               IF NOT "IX_HBW_SwitchCantileverFront_I5" AND "IX_HBW_SwitchCantileverBack_I6" THEN
                   IF "gtyp_VGR".x_HBW_Storage THEN
                       "gtyp_HBW".Rack_Workpiece[#li_Counter_Act_Ver, #li_Counter_Act_Hor].s_id := '';
                   ELSIF "gtyp_VGR".x_HBW_Outsource THEN
                       "gtyp_Interface_Dashboard".Subscribe.State_HBW.x_active := TRUE;
                       "gtyp_HBW".History := "gtyp_HBW".Rack_History[#li_Counter_Act_Ver, #li_Counter_Act_Hor].History;
                       "gtyp_HBW".Workpiece := "gtyp_HBW".Rack_Workpiece[#li_Counter_Act_Ver, #li_Counter_Act_Hor];
                       #li_Return_LDT := RD_SYS_T(#ldt_MQTT);
                       "gtyp_HBW".History[4].i_code := 400;
                       "gtyp_HBW".History[4].ldt_ts := DT_TO_LDT(#ldt_MQTT);

                       "gtyp_HBW".Rack_Workpiece[#li_Counter_Act_Ver, #li_Counter_Act_Hor].s_id := '';
                       "gtyp_HBW".Rack_Workpiece[#li_Counter_Act_Ver, #li_Counter_Act_Hor].s_state := '';
                       "gtyp_HBW".Rack_Workpiece[#li_Counter_Act_Ver, #li_Counter_Act_Hor].s_type := '';
                       FOR #li_Counter := 1 TO 8 DO
                           "gtyp_HBW".Rack_History[#li_Counter_Act_Ver, #li_Counter_Act_Hor].History[#li_Counter].i_code := 0;
                           "gtyp_HBW".Rack_History[#li_Counter_Act_Ver, #li_Counter_Act_Hor].History[#li_Counter].ldt_ts := DT#1990-01-01-00:00:00;
                       END_FOR;
                   END_IF;
                   "QX_HBW_M4_CantileverBackward_Q8" := FALSE;
                   "QX_HBW_M4_CantileverForward_Q7" := FALSE;
                   #li_StepCase := 110;
               END_IF;

           110: // homing vertical/horizontal axis

               "gtyp_HBW".Horizontal_Axis.x_Reference := TRUE;

               "gtyp_HBW".Vertical_Axis.di_Target_Position := "gtyp_HBW".di_PosBelt_Vertical - "gtyp_HBW".di_Offset_Pos_Belt_Vertical;
               "gtyp_HBW".Vertical_Axis.x_Start_Positioning := TRUE;

               IF ("gtyp_HBW".Vertical_Axis.di_Actual_Position <= ("gtyp_HBW".di_PosBelt_Vertical - "gtyp_HBW".di_Offset_Pos_Belt_Vertical + "gtyp_HBW".Vertical_Axis.Config.di_Pos_Window))
                   AND ("gtyp_HBW".Vertical_Axis.di_Actual_Position >= ("gtyp_HBW".di_PosBelt_Vertical - "gtyp_HBW".di_Offset_Pos_Belt_Vertical - "gtyp_HBW".Vertical_Axis.Config.di_Pos_Window))
                   AND "gtyp_HBW".Vertical_Axis.x_Position_Reached THEN
                   "gtyp_HBW".Vertical_Axis.x_Start_Positioning := FALSE;
               END_IF;

               IF NOT "gtyp_HBW".Horizontal_Axis.x_Referenced THEN
                   #li_StepCase := 120;
               END_IF;

           120: //homed vertical/horizontal axis

               IF "gtyp_HBW".Horizontal_Axis.x_Referenced THEN
                   "gtyp_HBW".Horizontal_Axis.x_Reference := FALSE;
               END_IF;

               IF ("gtyp_HBW".Vertical_Axis.di_Actual_Position <= ("gtyp_HBW".di_PosBelt_Vertical - "gtyp_HBW".di_Offset_Pos_Belt_Vertical + "gtyp_HBW".Vertical_Axis.Config.di_Pos_Window))
                   AND ("gtyp_HBW".Vertical_Axis.di_Actual_Position >= ("gtyp_HBW".di_PosBelt_Vertical - "gtyp_HBW".di_Offset_Pos_Belt_Vertical - "gtyp_HBW".Vertical_Axis.Config.di_Pos_Window))
                   AND "gtyp_HBW".Vertical_Axis.x_Position_Reached THEN
                   "gtyp_HBW".Vertical_Axis.x_Start_Positioning := FALSE;
               END_IF;

               IF "gtyp_HBW".Horizontal_Axis.x_Referenced
                   AND ("gtyp_HBW".Vertical_Axis.di_Actual_Position <= ("gtyp_HBW".di_PosBelt_Vertical - "gtyp_HBW".di_Offset_Pos_Belt_Vertical + "gtyp_HBW".Vertical_Axis.Config.di_Pos_Window))
                   AND ("gtyp_HBW".Vertical_Axis.di_Actual_Position >= ("gtyp_HBW".di_PosBelt_Vertical - "gtyp_HBW".di_Offset_Pos_Belt_Vertical - "gtyp_HBW".Vertical_Axis.Config.di_Pos_Window))
                   AND "gtyp_HBW".Vertical_Axis.x_Position_Reached THEN
                   "gtyp_HBW".Horizontal_Axis.x_Reference := FALSE;
                   "gtyp_HBW".Vertical_Axis.x_Start_Positioning := FALSE;
                   #li_StepCase := 130;
               END_IF;

           130: // Position vertical+offset/horizontal Belt
               "gtyp_HBW".Horizontal_Axis.di_Target_Position := "gtyp_HBW".di_PosBelt_Horizontal;
               "gtyp_HBW".Horizontal_Axis.x_Start_Positioning := TRUE;

               IF ("gtyp_HBW".Horizontal_Axis.di_Actual_Position <= ("gtyp_HBW".di_PosBelt_Horizontal + "gtyp_HBW".Horizontal_Axis.Config.di_Pos_Window))
                   AND ("gtyp_HBW".Horizontal_Axis.di_Actual_Position >= ("gtyp_HBW".di_PosBelt_Horizontal - "gtyp_HBW".Horizontal_Axis.Config.di_Pos_Window))
                   AND "gtyp_HBW".Horizontal_Axis.x_Position_Reached THEN
                   "gtyp_HBW".Horizontal_Axis.x_Start_Positioning := FALSE;
               END_IF;

               IF ("gtyp_HBW".Horizontal_Axis.di_Actual_Position <= ("gtyp_HBW".di_PosBelt_Horizontal + "gtyp_HBW".Horizontal_Axis.Config.di_Pos_Window))
                   AND ("gtyp_HBW".Horizontal_Axis.di_Actual_Position >= ("gtyp_HBW".di_PosBelt_Horizontal - "gtyp_HBW".Horizontal_Axis.Config.di_Pos_Window))
                   AND "gtyp_HBW".Horizontal_Axis.x_Position_Reached THEN
                   "gtyp_HBW".Horizontal_Axis.x_Start_Positioning := FALSE;
                   #li_StepCase := 140;
               END_IF;

           140: // Position cantilever Forward Belt

               "QX_HBW_M4_CantileverBackward_Q8" := FALSE;
               "QX_HBW_M4_CantileverForward_Q7" := TRUE;

               #lx_Time_Error := TRUE;

               IF "IX_HBW_SwitchCantileverFront_I5" AND NOT "IX_HBW_SwitchCantileverBack_I6" THEN
                   "QX_HBW_M4_CantileverBackward_Q8" := FALSE;
                   "QX_HBW_M4_CantileverForward_Q7" := FALSE;
                   #lx_Time_Error := FALSE;
                   #li_StepCase := 150;
               END_IF;

               // runtime error
               IF #lfb_TON_Error.Q THEN
                   #li_Lights := 4;
                   #lx_Time_Error := FALSE;
                   "QX_HBW_M1_ConveyorBeltBackward_Q2" := FALSE;
                   "QX_HBW_M1_ConveyorBeltForward_Q1" := FALSE;
                   "gtyp_Interface_Dashboard".Subscribe.State_HBW.x_active := FALSE;
                   "gtyp_HBW".x_Error := TRUE;
                   #li_StepCase := 0;
               END_IF;

           150: // Position vertical Belt
               "gtyp_HBW".Vertical_Axis.di_Target_Position := "gtyp_HBW".di_PosBelt_Vertical;
               "gtyp_HBW".Vertical_Axis.x_Start_Positioning := TRUE;

               IF ("gtyp_HBW".Vertical_Axis.di_Actual_Position <= ("gtyp_HBW".di_PosBelt_Vertical + "gtyp_HBW".Vertical_Axis.Config.di_Pos_Window))
                   AND ("gtyp_HBW".Vertical_Axis.di_Actual_Position >= ("gtyp_HBW".di_PosBelt_Vertical - "gtyp_HBW".Vertical_Axis.Config.di_Pos_Window))
                   AND "gtyp_HBW".Vertical_Axis.x_Position_Reached THEN
                   "gtyp_HBW".Vertical_Axis.x_Start_Positioning := FALSE;
                   #li_StepCase := 160;
               END_IF;

           160: // Start Conveyor Belt Forward

               #lx_Time_Error := TRUE;

               IF NOT "IX_HBW_LightBarrierInside_I2" THEN
                   "QX_HBW_M1_ConveyorBeltBackward_Q2" := FALSE;
                   "QX_HBW_M1_ConveyorBeltForward_Q1" := TRUE;
                   #lx_Time_Error := FALSE;
                   #li_StepCase := 170;
               END_IF;

               // runtime error
               IF #lfb_TON_Error.Q THEN
                   #li_Lights := 4;
                   #lx_Time_Error := FALSE;
                   "QX_HBW_M1_ConveyorBeltBackward_Q2" := FALSE;
                   "QX_HBW_M1_ConveyorBeltForward_Q1" := FALSE;
                   "gtyp_Interface_Dashboard".Subscribe.State_HBW.x_active := FALSE;
                   "gtyp_HBW".x_Error := TRUE;
                   #li_StepCase := 0;
               END_IF;

           170: //Run-on time reached Conveyor Belt Outside

               #lx_Time_Error := TRUE;

               IF #lfb_TON_ConveyerBelt_Out.Q THEN
                   "QX_HBW_M1_ConveyorBeltBackward_Q2" := FALSE;
                   "QX_HBW_M1_ConveyorBeltForward_Q1" := FALSE;
                   "gtyp_HBW".x_HBW_Container_Available := TRUE;
                   #lx_Time_Error := FALSE;
                   #li_StepCase := 180;
               END_IF;

               // runtime error
               IF #lfb_TON_Error.Q THEN
                   #li_Lights := 4;
                   #lx_Time_Error := FALSE;
                   "QX_HBW_M1_ConveyorBeltBackward_Q2" := FALSE;
                   "QX_HBW_M1_ConveyorBeltForward_Q1" := FALSE;
                   "gtyp_Interface_Dashboard".Subscribe.State_HBW.x_active := FALSE;
                   "gtyp_HBW".x_Error := TRUE;
                   #li_StepCase := 0;
               END_IF;

           180: // VGR picked up - outsource

               #li_Lights := 1;

               IF "gtyp_VGR".x_HBW_PickedUp AND "gtyp_VGR".x_HBW_Outsource THEN
                   "gtyp_VGR".Workpiece := "gtyp_HBW".Workpiece;
                   "gtyp_VGR".History := "gtyp_HBW".History;
                   "gtyp_HBW".Workpiece.s_id := '0';
                   "gtyp_HBW".Workpiece.s_state := '';
                   "gtyp_HBW".Workpiece.s_type := '';
                   FOR #li_Counter := 1 TO 8 DO
                       "gtyp_HBW".History[#li_Counter].i_code := 0;
                       "gtyp_HBW".History[#li_Counter].ldt_ts := DT#1990-01-01-00:00:00;
                   END_FOR;
                   "gtyp_HBW".x_HBW_Container_Available := FALSE;
                   "gtyp_HBW".x_HBW_PickedUp_Accepted := TRUE;

                   "gtyp_Interface_Dashboard".Subscribe.State_HBW.x_active := FALSE;

                   #li_Lights := 2;
                   #li_StepCase := 190;
                   // VGR discard - storage
               ELSIF "gtyp_VGR".x_HBW_Discards AND "gtyp_VGR".x_HBW_Storage THEN
                   "gtyp_Interface_Dashboard".Subscribe.State_HBW.x_active := TRUE;
                   "gtyp_HBW".Workpiece := "gtyp_VGR".Workpiece;
                   "gtyp_HBW".History := "gtyp_VGR".History;
                   "gtyp_HBW".x_HBW_Container_Available := FALSE;
                   "gtyp_HBW".x_HBW_Discards_Accepted := TRUE;
                   #lx_Storage := true;

                   #li_Lights := 2;
                   #li_StepCase := 190;
               END_IF;

           190: // Start Conveyor Belt Back

               IF NOT "gtyp_VGR".x_HBW_Discards AND NOT "gtyp_VGR".x_HBW_PickedUp THEN
                   "QX_HBW_M1_ConveyorBeltBackward_Q2" := TRUE;
                   "QX_HBW_M1_ConveyorBeltForward_Q1" := FALSE;
                   #li_StepCase := 200;
               END_IF;

           200:  // Conveyor Belt inside reached

               #lx_Time_Error := TRUE;

               IF NOT "IX_HBW_LightBarrierInside_I2" THEN
                   "QX_HBW_M1_ConveyorBeltBackward_Q2" := FALSE;
                   "QX_HBW_M1_ConveyorBeltForward_Q1" := FALSE;
                   #lx_Time_Error := FALSE;
                   #li_StepCase := 210;
               END_IF;

               // runtime error
               IF #lfb_TON_Error.Q THEN
                   #li_Lights := 4;
                   #lx_Time_Error := FALSE;
                   "QX_HBW_M1_ConveyorBeltBackward_Q2" := FALSE;
                   "QX_HBW_M1_ConveyorBeltForward_Q1" := FALSE;
                   "gtyp_Interface_Dashboard".Subscribe.State_HBW.x_active := FALSE;
                   "gtyp_HBW".x_Error := TRUE;
                   #li_StepCase := 0;
               END_IF;

           210: // Position vertical+offset Belt

               "gtyp_HBW".Vertical_Axis.di_Target_Position := "gtyp_HBW".di_PosBelt_Vertical - "gtyp_HBW".di_Offset_Pos_Belt_Vertical;
               "gtyp_HBW".Vertical_Axis.x_Start_Positioning := TRUE;

               IF ("gtyp_HBW".Vertical_Axis.di_Actual_Position <= ("gtyp_HBW".di_PosBelt_Vertical - "gtyp_HBW".di_Offset_Pos_Belt_Vertical + "gtyp_HBW".Vertical_Axis.Config.di_Pos_Window))
                   AND ("gtyp_HBW".Vertical_Axis.di_Actual_Position >= ("gtyp_HBW".di_PosBelt_Vertical - "gtyp_HBW".di_Offset_Pos_Belt_Vertical - "gtyp_HBW".Vertical_Axis.Config.di_Pos_Window))
                   AND "gtyp_HBW".Vertical_Axis.x_Position_Reached THEN
                   "gtyp_HBW".Vertical_Axis.x_Start_Positioning := FALSE;
               END_IF;

               IF ("gtyp_HBW".Vertical_Axis.di_Actual_Position <= ("gtyp_HBW".di_PosBelt_Vertical - "gtyp_HBW".di_Offset_Pos_Belt_Vertical + "gtyp_HBW".Vertical_Axis.Config.di_Pos_Window))
                   AND ("gtyp_HBW".Vertical_Axis.di_Actual_Position >= ("gtyp_HBW".di_PosBelt_Vertical - "gtyp_HBW".di_Offset_Pos_Belt_Vertical - "gtyp_HBW".Vertical_Axis.Config.di_Pos_Window))
                   AND "gtyp_HBW".Vertical_Axis.x_Position_Reached THEN
                   "gtyp_HBW".Vertical_Axis.x_Start_Positioning := FALSE;
                   #li_StepCase := 220;
               END_IF;

           220: // Position Cantilever back Belt   
               "QX_HBW_M4_CantileverBackward_Q8" := TRUE;
               "QX_HBW_M4_CantileverForward_Q7" := FALSE;

               IF NOT "IX_HBW_SwitchCantileverFront_I5" AND "IX_HBW_SwitchCantileverBack_I6" THEN
                   "QX_HBW_M4_CantileverBackward_Q8" := FALSE;
                   "QX_HBW_M4_CantileverForward_Q7" := FALSE;
                   #li_StepCase := 230;
               END_IF;

           230: // Position vertical+offset/horizontal HBW
               "gtyp_HBW".Horizontal_Axis.di_Target_Position := #ldi_PosRack_Horizontal;
               "gtyp_HBW".Horizontal_Axis.x_Start_Positioning := TRUE;
               "gtyp_HBW".Vertical_Axis.di_Target_Position := #ldi_PosRack_Vertical - "gtyp_HBW".di_Offset_Pos_Rack_Vertical;
               "gtyp_HBW".Vertical_Axis.x_Start_Positioning := TRUE;

               IF ("gtyp_HBW".Horizontal_Axis.di_Actual_Position <= (#ldi_PosRack_Horizontal + "gtyp_HBW".Horizontal_Axis.Config.di_Pos_Window))
                   AND ("gtyp_HBW".Horizontal_Axis.di_Actual_Position >= (#ldi_PosRack_Horizontal - "gtyp_HBW".Horizontal_Axis.Config.di_Pos_Window))
                   AND "gtyp_HBW".Horizontal_Axis.x_Position_Reached THEN
                   "gtyp_HBW".Horizontal_Axis.x_Start_Positioning := FALSE;
               END_IF;

               IF ("gtyp_HBW".Vertical_Axis.di_Actual_Position <= (#ldi_PosRack_Vertical - "gtyp_HBW".di_Offset_Pos_Rack_Vertical + "gtyp_HBW".Vertical_Axis.Config.di_Pos_Window))
                   AND ("gtyp_HBW".Vertical_Axis.di_Actual_Position >= (#ldi_PosRack_Vertical - "gtyp_HBW".di_Offset_Pos_Rack_Vertical - "gtyp_HBW".Vertical_Axis.Config.di_Pos_Window))
                   AND "gtyp_HBW".Vertical_Axis.x_Position_Reached THEN
                   "gtyp_HBW".Vertical_Axis.x_Start_Positioning := FALSE;
               END_IF;

               IF ("gtyp_HBW".Horizontal_Axis.di_Actual_Position <= (#ldi_PosRack_Horizontal + "gtyp_HBW".Horizontal_Axis.Config.di_Pos_Window))
                   AND ("gtyp_HBW".Horizontal_Axis.di_Actual_Position >= (#ldi_PosRack_Horizontal - "gtyp_HBW".Horizontal_Axis.Config.di_Pos_Window))
                   AND "gtyp_HBW".Horizontal_Axis.x_Position_Reached
                   AND ("gtyp_HBW".Vertical_Axis.di_Actual_Position <= (#ldi_PosRack_Vertical - "gtyp_HBW".di_Offset_Pos_Rack_Vertical + "gtyp_HBW".Vertical_Axis.Config.di_Pos_Window))
                   AND ("gtyp_HBW".Vertical_Axis.di_Actual_Position >= (#ldi_PosRack_Vertical - "gtyp_HBW".di_Offset_Pos_Rack_Vertical - "gtyp_HBW".Vertical_Axis.Config.di_Pos_Window))
                   AND "gtyp_HBW".Vertical_Axis.x_Position_Reached THEN
                   "gtyp_HBW".Horizontal_Axis.x_Start_Positioning := FALSE;
                   "gtyp_HBW".Vertical_Axis.x_Start_Positioning := FALSE;
                   #li_StepCase := 240;
               END_IF;

           240: // Position Cantilever Forward HBW

               "QX_HBW_M4_CantileverBackward_Q8" := FALSE;
               "QX_HBW_M4_CantileverForward_Q7" := TRUE;

               IF "IX_HBW_SwitchCantileverFront_I5" AND NOT "IX_HBW_SwitchCantileverBack_I6" THEN
                   "QX_HBW_M4_CantileverBackward_Q8" := FALSE;
                   "QX_HBW_M4_CantileverForward_Q7" := FALSE;
                   #li_StepCase := 250;
               END_IF;

           250: // Position vertical HBW
               "gtyp_HBW".Vertical_Axis.di_Target_Position := #ldi_PosRack_Vertical;
               "gtyp_HBW".Vertical_Axis.x_Start_Positioning := TRUE;

               IF ("gtyp_HBW".Vertical_Axis.di_Actual_Position <= (#ldi_PosRack_Vertical + "gtyp_HBW".Vertical_Axis.Config.di_Pos_Window))
                   AND ("gtyp_HBW".Vertical_Axis.di_Actual_Position >= (#ldi_PosRack_Vertical - "gtyp_HBW".Vertical_Axis.Config.di_Pos_Window))
                   AND "gtyp_HBW".Vertical_Axis.x_Position_Reached THEN
                   IF #lx_Storage THEN
                       #li_Return_LDT := RD_SYS_T(#ldt_MQTT);
                       "gtyp_HBW".History[3].i_code := 300;
                       "gtyp_HBW".History[3].ldt_ts := DT_TO_LDT(#ldt_MQTT);
                       "gtyp_HBW".Rack_Workpiece[#li_Counter_Act_Ver, #li_Counter_Act_Hor] := "gtyp_HBW".Workpiece;
                       "gtyp_HBW".Rack_History[#li_Counter_Act_Ver, #li_Counter_Act_Hor].History := "gtyp_HBW".History;
                       "gtyp_Interface_Dashboard".Subscribe.State_HBW.x_active := FALSE;
                   ELSE
                       "gtyp_HBW".Rack_Workpiece[#li_Counter_Act_Ver, #li_Counter_Act_Hor].s_id := '0';
                   END_IF;
                   "gtyp_HBW".Vertical_Axis.x_Start_Positioning := FALSE;
                   #li_StepCase := 260;
               END_IF;

           260: // Position Cantilever Backward HBW

               "QX_HBW_M4_CantileverBackward_Q8" := TRUE;
               "QX_HBW_M4_CantileverForward_Q7" := FALSE;

               IF NOT "IX_HBW_SwitchCantileverFront_I5" AND "IX_HBW_SwitchCantileverBack_I6" THEN
                   "QX_HBW_M4_CantileverBackward_Q8" := FALSE;
                   "QX_HBW_M4_CantileverForward_Q7" := FALSE;
                   #li_StepCase := 0;
                   #lx_Storage := FALSE;
               END_IF;
               // Statement section ELSE    
           ELSE
               ;
       END_CASE;

       //Reset the information in the high-bay warehouse
       IF "gtyp_Setup".x_Clean_Rack_HBW THEN
           FOR #li_Counter_Hor := 1 TO 3 DO
               FOR #li_Counter_Ver := 1 TO 3 DO
                   "gtyp_HBW".Rack_Workpiece[#li_Counter_Ver, #li_Counter_Hor].s_id := '0';
                   "gtyp_HBW".Rack_Workpiece[#li_Counter_Ver, #li_Counter_Hor].s_state := '';
                   "gtyp_HBW".Rack_Workpiece[#li_Counter_Ver, #li_Counter_Hor].s_type := '';
                   FOR #li_Counter := 1 TO 8 DO
                       "gtyp_HBW".Rack_History[#li_Counter_Ver, #li_Counter_Hor].History[#li_Counter].i_code := 0;
                       "gtyp_HBW".Rack_History[#li_Counter_Ver, #li_Counter_Hor].History[#li_Counter].ldt_ts := DT#1990-01-01-00:00:00;
                   END_FOR;
               END_FOR;
           END_FOR;
           "gtyp_Setup".x_Clean_Rack_HBW := FALSE;
       END_IF;

       // reload PWM
       "QW_HBW_PWM_ConveyorBelt_M1" := "gtyp_HBW"."i_PWM_ConveyorBelt";
       "QW_HBW_PWM_Cantilever_M4" := "gtyp_HBW"."i_PWM_Cantilever";
   ELSE
       FOR #li_Counter_Hor := 1 TO 3 DO
           FOR #li_Counter_Ver := 1 TO 3 DO
               IF "gtyp_HBW".Rack_Workpiece[#li_Counter_Ver, #li_Counter_Hor].s_id = '' THEN
                   "gtyp_HBW".Rack_Workpiece[#li_Counter_Ver, #li_Counter_Hor].s_id := '0';
                   "gtyp_HBW".Rack_Workpiece[#li_Counter_Ver, #li_Counter_Hor].s_state := '';
                   "gtyp_HBW".Rack_Workpiece[#li_Counter_Ver, #li_Counter_Hor].s_type := '';
                   FOR #li_Counter := 1 TO 8 DO
                       "gtyp_HBW".Rack_History[#li_Counter_Ver, #li_Counter_Hor].History[#li_Counter].i_code := 0;
                       "gtyp_HBW".Rack_History[#li_Counter_Ver, #li_Counter_Hor].History[#li_Counter].ldt_ts := DT#1990-01-01-00:00:00;
                   END_FOR;
               END_IF;
           END_FOR;
       END_FOR;

       "gtyp_HBW".x_Start_Park_Position := FALSE;
       "gtyp_HBW".x_Park_Position_Reached := FALSE;
       "gtyp_HBW".x_HBW_PickedUp_Accepted := FALSE;
       "gtyp_HBW".x_HBW_Discards_Accepted := FALSE;
       "gtyp_HBW".x_HBW_PickUp_Ready := FALSE;
       "gtyp_HBW".x_HBW_Container_Available := FALSE;
       "gtyp_HBW".x_Error := FALSE;

       #li_Lights := 1;
       #lx_Start_TON_Fill_HBW := TRUE;
       #lx_Init := TRUE;
   END_IF;
END_FUNCTION_BLOCK

FUNCTION_BLOCK "PRG_MPO_Ablauf"   // FB17, SCL
TITLE = Program Ablauf MPO
{ S7_Optimized_Access := 'TRUE' }
AUTHOR : A.Schaefer
VERSION : 0.0
   VAR
      lx_Init : Bool;
      lx_Start_TON_Wait : Bool;
      lx_Time_Error : Bool;
      lt_TON_Wait : Time;
      lx_Start_TON_State : Bool;
      ldt_MQTT : Date_And_Time;
      li_Return_LDT : Int;
      li_StepCase : Int;
      li_Lights : Int;
      li_Lights_old : Int;
      li_Counter : Int;
      lfb_blinker : "FB_Blinker";
      lfb_TOF_ConveyerBelt_Out : TOF_TIME;
      lfb_TON_Wait : TON_TIME;
      lfb_TON_Error : TON_TIME;
      lfb_TON_State : TON_TIME;
      lfb_F_Trig_ConveyerBelt : F_TRIG;
   END_VAR
BEGIN
   IF #lx_Init THEN

       // wait time state
       #lfb_TON_State(IN := NOT #lx_Start_TON_State,
                      PT := T#2s);

       // runtime monitoring error
       #lfb_TON_Error(IN := #lx_Time_Error,
                      PT := T#30s);

       // state of the MPO cyclically transmitted to the cloud
       IF (#lfb_TON_State.Q OR (#li_Lights <> #li_Lights_old)) AND NOT #lx_Start_TON_State THEN
           #li_Lights_old := #li_Lights;
           #lx_Start_TON_State := TRUE;
           #li_Return_LDT := RD_SYS_T(#ldt_MQTT);
           "gtyp_Interface_Dashboard".Subscribe.State_MPO.ldt_ts := DT_TO_LDT(#ldt_MQTT);
           "gtyp_Interface_Dashboard".Subscribe.State_MPO.i_code := #li_Lights;
           "gtyp_Interface_Dashboard".Subscribe.State_MPO.s_description := '';
           "gtyp_Interface_Dashboard".Subscribe.State_MPO.s_station := 'mpo';
           "gtyp_Interface_Dashboard".Subscribe.State_MPO.s_target := '';
       END_IF;

       // restart wait time state
       IF NOT #lfb_TON_State.Q AND #lx_Start_TON_State THEN
           #lx_Start_TON_State := FALSE;
       END_IF;

       // FB TON Wait
       #lfb_TON_Wait(IN := #lx_Start_TON_Wait,
                     PT := #lt_TON_Wait);

       // falling edge light barrier end of Conveyor Belt
       #lfb_F_Trig_ConveyerBelt(CLK := NOT "IX_MPO_LightBarrierEndOfConBelt_I3");

       //Run-on time Conveyer Belt
       #lfb_TOF_ConveyerBelt_Out(IN := #lfb_F_Trig_ConveyerBelt.Q,
                                 PT := T#5000ms);

       // FB blinker intervall 1s
       #lfb_blinker(int_periodendauer := T#1000ms);

       // step chain HBW
       CASE #li_StepCase OF

           0:  // init
               #lx_Start_TON_Wait := FALSE;
               #lx_Time_Error := FALSE;

               IF NOT "gtyp_MPO".x_Error AND NOT "gtyp_MPO".x_Start_Park_Position THEN
                   #li_StepCase := 10;
               END_IF;

           10: // turn-on Compressor and turn off oven light 
               #li_Lights := 2;
               "QX_MPO_LightOven_Q9" := FALSE;
               "QX_MPO_Compressor_Q10" := TRUE;

               #lx_Start_TON_Wait := TRUE;
               #lt_TON_Wait := T#500ms;

               IF #lfb_TON_Wait.Q THEN
                   #lx_Start_TON_Wait := FALSE;
                   #li_StepCase := 20;
               END_IF;

           20:  // Open oven door 
               "QX_MPO_ValveOvenDoor_Q13" := TRUE;
               "QX_MPO_ValveLowering_Q12" := FALSE;

               #lx_Start_TON_Wait := TRUE;
               #lt_TON_Wait := T#2000ms;

               IF #lfb_TON_Wait.Q THEN
                   #lx_Start_TON_Wait := FALSE;
                   #li_StepCase := 30;
               END_IF;

           30: // Position oven feeder retract
               IF "IX_MPO_RefSwitchOvenFeederOutside_I7" OR NOT "IX_MPO_RefSwitchOvenFeederInside_I6" THEN
                   "QX_MPO_M4_OvenFeederRetract_Q5" := TRUE;
                   "QX_MPO_M4_OvenFeederExtend_Q6" := FALSE;
               ELSIF NOT "IX_MPO_RefSwitchOvenFeederOutside_I7" AND "IX_MPO_RefSwitchOvenFeederInside_I6" THEN
                   "QX_MPO_M4_OvenFeederRetract_Q5" := FALSE;
                   "QX_MPO_M4_OvenFeederExtend_Q6" := FALSE;
                   #li_StepCase := 40;
               END_IF;

           40:  // Close door, Position Vacuum Towards Turn Table and vacuum off

               "QX_MPO_ValveOvenDoor_Q13" := FALSE;

               "QX_MPO_M5_VacuumTowardsTurnTable_Q8" := TRUE;
               "QX_MPO_M5_VacuumTowardsOven_Q7" := FALSE;
               "QX_MPO_ValveVacuum_Q11" := FALSE;

               IF "IX_MPO_RefSwitchVac_PosOven_I8" OR NOT "IX_MPO_RefSwitchVac_PosTurnTable_I5" THEN
                   "QX_MPO_M5_VacuumTowardsTurnTable_Q8" := TRUE;
                   "QX_MPO_M5_VacuumTowardsOven_Q7" := FALSE;
               ELSIF NOT "IX_MPO_RefSwitchVac_PosOven_I8" AND "IX_MPO_RefSwitchVac_PosTurnTable_I5" THEN
                   "QX_MPO_M5_VacuumTowardsTurnTable_Q8" := FALSE;
                   "QX_MPO_M5_VacuumTowardsOven_Q7" := FALSE;
                   #li_StepCase := 50;
               END_IF
               ;

           50: // saw, valve feeder conveyor belt off
               "QX_MPO_M3_Saw_Q4" := FALSE;
               "QX_MPO_ValveFeeder_Q14" := FALSE;
               "QX_MPO_M2_ConveyorBeltForward_Q3" := FALSE;

               IF "IX_MPO_RefSwitchTurnTable_PosSaw_I4" OR "IX_MPO_RefSwitchTurnTable_PosBelt_I2" OR NOT "IX_MPO_RefSwitchTurnTable_PosVac_I1" THEN
                   "QX_MPO_M1_TurnTableClockwise_Q1" := FALSE;
                   "QX_MPO_M1_TurnTableCounterclockwise_Q2" := TRUE;
               ELSIF NOT "IX_MPO_RefSwitchTurnTable_PosSaw_I4" AND NOT "IX_MPO_RefSwitchTurnTable_PosBelt_I2" AND "IX_MPO_RefSwitchTurnTable_PosVac_I1" THEN
                   "QX_MPO_M1_TurnTableClockwise_Q1" := FALSE;
                   "QX_MPO_M1_TurnTableCounterclockwise_Q2" := FALSE;
                   "QX_MPO_Compressor_Q10" := FALSE;
                   #li_StepCase := 60;
               END_IF;

           60: // wait for request discard form VGR
               #li_Lights := 1;
               IF "gtyp_VGR".x_MPO_Req_Discard THEN
                   #li_Lights := 2;
                   "QX_MPO_Compressor_Q10" := TRUE;
                   #li_StepCase := 70;
               END_IF;

           70: // wait sequence
               #lx_Start_TON_Wait := TRUE;
               #lt_TON_Wait := T#500ms;

               IF #lfb_TON_Wait.Q THEN
                   #lx_Start_TON_Wait := FALSE;
                   #li_StepCase := 80;
               END_IF;

           80: // open oven door
               "QX_MPO_ValveOvenDoor_Q13" := TRUE;

               #lx_Start_TON_Wait := TRUE;
               #lt_TON_Wait := T#2000ms;

               IF #lfb_TON_Wait.Q THEN
                   #lx_Start_TON_Wait := FALSE;
                   #li_StepCase := 90;
               END_IF;

           90: // oven feeder extend
               "QX_MPO_M4_OvenFeederRetract_Q5" := FALSE;
               "QX_MPO_M4_OvenFeederExtend_Q6" := TRUE;

               IF "IX_MPO_RefSwitchOvenFeederOutside_I7" AND NOT "IX_MPO_RefSwitchOvenFeederInside_I6" THEN
                   "QX_MPO_M4_OvenFeederRetract_Q5" := FALSE;
                   "QX_MPO_M4_OvenFeederExtend_Q6" := FALSE;
                   "gtyp_MPO".x_MPO_Discards_Accepted := FALSE;
                   "gtyp_MPO".x_Discard_Ready := TRUE;
                   #li_StepCase := 100;
               END_IF;

           100: // wait for VGR discard workpiece

               #lx_Time_Error := TRUE;

               IF "gtyp_VGR".x_MPO_Discards AND NOT "IX_MPO_LightBarrierOven_I9" THEN
                   "gtyp_Interface_Dashboard".Subscribe.State_MPO.x_active := TRUE;
                   "gtyp_MPO".History := "gtyp_VGR".History;
                   "gtyp_MPO".Workpiece := "gtyp_VGR".Workpiece;
                   "gtyp_MPO".x_Discard_Ready := FALSE;
                   "gtyp_MPO".x_MPO_Discards_Accepted := TRUE;
                   #lx_Time_Error := FALSE;
                   #li_StepCase := 105;
               END_IF;

               // runtime error
               IF #lfb_TON_Error.Q THEN
                   #li_Lights := 4;
                   #lx_Time_Error := FALSE;
                   "gtyp_Interface_Dashboard".Subscribe.State_Order.ldt_ts := DT_TO_LDT(#ldt_MQTT);
                   "gtyp_Interface_Dashboard".Subscribe.State_Order.s_state := 'WAITING_FOR_ORDER';
                   "gtyp_Interface_Dashboard".Subscribe.State_Order.s_type := '';
                   "gtyp_Interface_Dashboard".Subscribe.State_MPO.x_active := FALSE;
                   "gtyp_MPO".x_Discard_Ready := FALSE;
                   "gtyp_MPO".x_MPO_Discards_Accepted := FALSE;
                   "gtyp_MPO".x_Error := TRUE;
                   #li_StepCase := 0;
               END_IF;

           105: // VGR outside oven feeder - oven feeder retract
               IF NOT "gtyp_VGR".x_MPO_Discards AND "IX_MPO_RefSwitchOvenFeederOutside_I7" AND NOT "IX_MPO_RefSwitchOvenFeederInside_I6" THEN
                   "gtyp_MPO".x_MPO_Discards_Accepted := FALSE;
                   "QX_MPO_M4_OvenFeederRetract_Q5" := TRUE;
                   "QX_MPO_M4_OvenFeederExtend_Q6" := FALSE;
                   #li_StepCase := 110;
               END_IF;

           110: // sensor oven feeder inside reached
               IF NOT "IX_MPO_RefSwitchOvenFeederOutside_I7" AND "IX_MPO_RefSwitchOvenFeederInside_I6" THEN
                   "QX_MPO_M4_OvenFeederRetract_Q5" := FALSE;
                   "QX_MPO_M4_OvenFeederExtend_Q6" := FALSE;
                   #li_StepCase := 120;
               END_IF;

           120: // close oven door
               "QX_MPO_ValveOvenDoor_Q13" := FALSE;

               #lx_Start_TON_Wait := TRUE;
               #lt_TON_Wait := T#2000ms;

               IF #lfb_TON_Wait.Q THEN
                   #lx_Start_TON_Wait := FALSE;
                   #li_StepCase := 130;
               END_IF;

           130: // processing time flashing interval
               "QX_MPO_LightOven_Q9" := #lfb_blinker.outx_blinker;

               IF NOT "gtyp_VGR".x_MPO_Discards THEN
                   #li_Return_LDT := RD_SYS_T(#ldt_MQTT);
                   "gtyp_MPO".History[5].i_code := 500;
                   "gtyp_MPO".History[5].ldt_ts := DT_TO_LDT(#ldt_MQTT);

                   "QX_MPO_M5_VacuumTowardsOven_Q7" := TRUE;
                   "QX_MPO_M5_VacuumTowardsTurnTable_Q8" := FALSE;

                   IF NOT "IX_MPO_RefSwitchVac_PosTurnTable_I5" AND "IX_MPO_RefSwitchVac_PosOven_I8" THEN
                       "QX_MPO_M5_VacuumTowardsOven_Q7" := FALSE;
                       "QX_MPO_M5_VacuumTowardsTurnTable_Q8" := FALSE;
                   END_IF;
               END_IF;

               #lx_Start_TON_Wait := TRUE;
               #lt_TON_Wait := T#4000ms;

               IF #lfb_TON_Wait.Q THEN
                   #lx_Start_TON_Wait := FALSE;
                   #li_StepCase := 140;
               END_IF;

           140: // open oven door
               "QX_MPO_LightOven_Q9" := FALSE;
               "QX_MPO_ValveOvenDoor_Q13" := TRUE;

               IF NOT "gtyp_VGR".x_MPO_Discards THEN
                   "QX_MPO_M5_VacuumTowardsOven_Q7" := TRUE;
                   "QX_MPO_M5_VacuumTowardsTurnTable_Q8" := FALSE;

                   IF NOT "IX_MPO_RefSwitchVac_PosTurnTable_I5" AND "IX_MPO_RefSwitchVac_PosOven_I8" THEN
                       "QX_MPO_M5_VacuumTowardsOven_Q7" := FALSE;
                       "QX_MPO_M5_VacuumTowardsTurnTable_Q8" := FALSE;
                   END_IF;
               END_IF;

               #lx_Start_TON_Wait := TRUE;
               #lt_TON_Wait := T#2000ms;

               IF #lfb_TON_Wait.Q THEN
                   #lx_Start_TON_Wait := FALSE;
                   #li_StepCase := 150;
               END_IF;

           150: // oven feeder extend

               "QX_MPO_M4_OvenFeederRetract_Q5" := FALSE;
               "QX_MPO_M4_OvenFeederExtend_Q6" := TRUE;

               IF NOT "gtyp_VGR".x_MPO_Discards THEN
                   "QX_MPO_M5_VacuumTowardsOven_Q7" := TRUE;
                   "QX_MPO_M5_VacuumTowardsTurnTable_Q8" := FALSE;

                   IF NOT "IX_MPO_RefSwitchVac_PosTurnTable_I5" AND "IX_MPO_RefSwitchVac_PosOven_I8" THEN
                       "QX_MPO_M5_VacuumTowardsOven_Q7" := FALSE;
                       "QX_MPO_M5_VacuumTowardsTurnTable_Q8" := FALSE;
                   END_IF;
               END_IF;

               IF "IX_MPO_RefSwitchOvenFeederOutside_I7" AND NOT "IX_MPO_RefSwitchOvenFeederInside_I6" THEN
                   "QX_MPO_M4_OvenFeederRetract_Q5" := FALSE;
                   "QX_MPO_M4_OvenFeederExtend_Q6" := FALSE;
               END_IF;

               IF "IX_MPO_RefSwitchOvenFeederOutside_I7" AND NOT "IX_MPO_RefSwitchOvenFeederInside_I6"
                   AND NOT "IX_MPO_RefSwitchVac_PosTurnTable_I5" AND "IX_MPO_RefSwitchVac_PosOven_I8" THEN
                   "QX_MPO_M5_VacuumTowardsOven_Q7" := FALSE;
                   "QX_MPO_M5_VacuumTowardsTurnTable_Q8" := FALSE;
                   "QX_MPO_M4_OvenFeederRetract_Q5" := FALSE;
                   "QX_MPO_M4_OvenFeederExtend_Q6" := FALSE;
                   #li_StepCase := 160;
               END_IF;

           160: // vacuum suction device down
               "QX_MPO_ValveLowering_Q12" := TRUE;

               #lx_Start_TON_Wait := TRUE;
               #lt_TON_Wait := T#1000ms;

               IF #lfb_TON_Wait.Q THEN
                   #lx_Start_TON_Wait := FALSE;
                   #li_StepCase := 170;
               END_IF;

           170: // vacuum suction device picks up the workpiece
               "QX_MPO_ValveVacuum_Q11" := TRUE;

               #lx_Start_TON_Wait := TRUE;
               #lt_TON_Wait := T#1000ms;

               IF #lfb_TON_Wait.Q THEN
                   #lx_Start_TON_Wait := FALSE;
                   #li_StepCase := 180;
               END_IF;

           180: // vacuum suction device up
               "QX_MPO_ValveLowering_Q12" := FALSE;

               #lx_Start_TON_Wait := TRUE;
               #lt_TON_Wait := T#1000ms;

               IF #lfb_TON_Wait.Q THEN
                   #lx_Start_TON_Wait := FALSE;
                   #li_StepCase := 190;
               END_IF;

           190: // oven feeder retract and vacuum towards turn table
               "QX_MPO_M4_OvenFeederRetract_Q5" := TRUE;
               "QX_MPO_M4_OvenFeederExtend_Q6" := FALSE;
               "QX_MPO_M5_VacuumTowardsOven_Q7" := FALSE;
               "QX_MPO_M5_VacuumTowardsTurnTable_Q8" := TRUE;

               IF "IX_MPO_RefSwitchVac_PosTurnTable_I5" AND NOT "IX_MPO_RefSwitchVac_PosOven_I8" THEN
                   "QX_MPO_M5_VacuumTowardsOven_Q7" := FALSE;
                   "QX_MPO_M5_VacuumTowardsTurnTable_Q8" := FALSE;
               END_IF;

               IF NOT "IX_MPO_RefSwitchOvenFeederOutside_I7" AND "IX_MPO_RefSwitchOvenFeederInside_I6" THEN
                   "QX_MPO_M4_OvenFeederRetract_Q5" := FALSE;
                   "QX_MPO_M4_OvenFeederExtend_Q6" := FALSE;
               END_IF;

               IF NOT "IX_MPO_RefSwitchOvenFeederOutside_I7" AND "IX_MPO_RefSwitchOvenFeederInside_I6"
                   AND "IX_MPO_RefSwitchVac_PosTurnTable_I5" AND NOT "IX_MPO_RefSwitchVac_PosOven_I8" THEN
                   "QX_MPO_M5_VacuumTowardsOven_Q7" := FALSE;
                   "QX_MPO_M5_VacuumTowardsTurnTable_Q8" := FALSE;
                   "QX_MPO_M4_OvenFeederRetract_Q5" := FALSE;
                   "QX_MPO_M4_OvenFeederExtend_Q6" := FALSE;
                   "QX_MPO_ValveOvenDoor_Q13" := FALSE;
                   #li_StepCase := 200;
               END_IF;

           200: // vacuum suction device down at turn table
               IF "IX_MPO_RefSwitchTurnTable_PosVac_I1" THEN
                   "QX_MPO_ValveLowering_Q12" := TRUE;

                   #lx_Start_TON_Wait := TRUE;
                   #lt_TON_Wait := T#2000ms;

                   IF #lfb_TON_Wait.Q THEN
                       #lx_Start_TON_Wait := FALSE;
                       #li_StepCase := 210;
                   END_IF;
               END_IF;

           210: // vacuum off
               "QX_MPO_ValveVacuum_Q11" := FALSE;

               #lx_Start_TON_Wait := TRUE;
               #lt_TON_Wait := T#2000ms;

               IF #lfb_TON_Wait.Q THEN
                   #lx_Start_TON_Wait := FALSE;
                   #li_StepCase := 220;
               END_IF;

           220: // vacuum suction device up
               "QX_MPO_ValveLowering_Q12" := FALSE;

               #lx_Start_TON_Wait := TRUE;
               #lt_TON_Wait := T#2000ms;

               IF #lfb_TON_Wait.Q THEN
                   #lx_Start_TON_Wait := FALSE;
                   #li_StepCase := 230;
               END_IF;

           230: // Position turn table saw
               IF NOT "IX_MPO_RefSwitchTurnTable_PosSaw_I4" AND NOT "IX_MPO_RefSwitchTurnTable_PosBelt_I2" AND "IX_MPO_RefSwitchTurnTable_PosVac_I1" THEN
                   "QX_MPO_M1_TurnTableClockwise_Q1" := TRUE;
                   "QX_MPO_M1_TurnTableCounterclockwise_Q2" := FALSE;
               ELSIF "IX_MPO_RefSwitchTurnTable_PosSaw_I4" OR "IX_MPO_RefSwitchTurnTable_PosBelt_I2" AND NOT "IX_MPO_RefSwitchTurnTable_PosVac_I1" THEN
                   "QX_MPO_M1_TurnTableClockwise_Q1" := FALSE;
                   "QX_MPO_M1_TurnTableCounterclockwise_Q2" := FALSE;
                   #li_StepCase := 240;
               END_IF;

           240: // Start sawing
               "QX_MPO_M3_Saw_Q4" := TRUE;

               #lx_Start_TON_Wait := TRUE;
               #lt_TON_Wait := T#4000ms;

               IF #lfb_TON_Wait.Q THEN
                   #li_Return_LDT := RD_SYS_T(#ldt_MQTT);
                   "gtyp_MPO".History[6].i_code := 600;
                   "gtyp_MPO".History[6].ldt_ts := DT_TO_LDT(#ldt_MQTT);

                   #lx_Start_TON_Wait := FALSE;
                   "QX_MPO_M3_Saw_Q4" := FALSE;
                   #li_StepCase := 250;
               END_IF;

           250: // Position turn table Pos Belt
               IF "IX_MPO_RefSwitchTurnTable_PosSaw_I4" AND NOT "IX_MPO_RefSwitchTurnTable_PosBelt_I2" AND NOT "IX_MPO_RefSwitchTurnTable_PosVac_I1" THEN
                   "QX_MPO_M1_TurnTableClockwise_Q1" := TRUE;
                   "QX_MPO_M1_TurnTableCounterclockwise_Q2" := FALSE;
               ELSIF NOT "IX_MPO_RefSwitchTurnTable_PosSaw_I4" AND "IX_MPO_RefSwitchTurnTable_PosBelt_I2" AND NOT "IX_MPO_RefSwitchTurnTable_PosVac_I1" THEN
                   "QX_MPO_M1_TurnTableClockwise_Q1" := FALSE;
                   "QX_MPO_M1_TurnTableCounterclockwise_Q2" := FALSE;
                   #li_StepCase := 260;
               END_IF;

           260: // put workpiece to belt
               "QX_MPO_ValveFeeder_Q14" := TRUE;

               #lx_Start_TON_Wait := TRUE;
               #lt_TON_Wait := T#1000ms;

               IF #lfb_TON_Wait.Q THEN
                   #lx_Start_TON_Wait := FALSE;
                   "QX_MPO_ValveFeeder_Q14" := FALSE;
                   "QX_MPO_Compressor_Q10" := FALSE;
                   #li_StepCase := 270;
               END_IF;

           270: // Position turn table Pos Vacuum
               IF "IX_MPO_RefSwitchTurnTable_PosSaw_I4" OR "IX_MPO_RefSwitchTurnTable_PosBelt_I2" OR NOT "IX_MPO_RefSwitchTurnTable_PosVac_I1" THEN
                   "QX_MPO_M1_TurnTableClockwise_Q1" := FALSE;
                   "QX_MPO_M1_TurnTableCounterclockwise_Q2" := TRUE;
               ELSIF NOT "IX_MPO_RefSwitchTurnTable_PosSaw_I4" AND NOT "IX_MPO_RefSwitchTurnTable_PosBelt_I2" AND "IX_MPO_RefSwitchTurnTable_PosVac_I1" THEN
                   "QX_MPO_M1_TurnTableClockwise_Q1" := FALSE;
                   "QX_MPO_M1_TurnTableCounterclockwise_Q2" := FALSE;
                   "QX_MPO_Compressor_Q10" := FALSE;
                   #li_StepCase := 280;
               END_IF;

           280: // Start conveyor belt
               "QX_MPO_M2_ConveyorBeltForward_Q3" := TRUE;

               #lx_Time_Error := TRUE;

               IF #lfb_TOF_ConveyerBelt_Out.Q THEN
                   "gtyp_SLD".History := "gtyp_MPO".History;
                   "gtyp_SLD".Workpiece := "gtyp_MPO".Workpiece;
                   "gtyp_MPO".Workpiece.s_id := '0';
                   "gtyp_MPO".Workpiece.s_state := '';
                   "gtyp_MPO".Workpiece.s_type := '';
                   FOR #li_Counter := 1 TO 8 DO
                       "gtyp_MPO".History[#li_Counter].i_code := 0;
                       "gtyp_MPO".History[#li_Counter].ldt_ts := DT#1990-01-01-00:00:00;
                   END_FOR;

                   "gtyp_Interface_Dashboard".Subscribe.State_MPO.x_active := FALSE;

                   #lx_Time_Error := FALSE;
                   #li_StepCase := 290;
               END_IF;

               // runtime error
               IF #lfb_TON_Error.Q THEN
                   #li_Lights := 4;
                   #lx_Time_Error := FALSE;
                   "QX_MPO_M2_ConveyorBeltForward_Q3" := FALSE;
                   "gtyp_Interface_Dashboard".Subscribe.State_MPO.x_active := FALSE;
                   "gtyp_MPO".x_Error := TRUE;
                   #li_StepCase := 0;
               END_IF;

           290: // wait for runtime on conveyor belt

               IF NOT #lfb_TOF_ConveyerBelt_Out.Q THEN
                   #lx_Start_TON_Wait := FALSE;
                   "QX_MPO_M2_ConveyorBeltForward_Q3" := FALSE;
                   #li_StepCase := 60;
               END_IF;
               // Statement section ELSE
           ELSE
               ;
       END_CASE;

       "QW_MPO_PWM_TurnTable_M1" := "gtyp_MPO"."i_PWM_TurnTable";
       "QW_MPO_PWM_Vacuum_M5" := "gtyp_MPO"."i_PWM_Vacuum";

   ELSE
       #li_Lights := 1;
       #lx_Init := TRUE;
       "gtyp_MPO".x_Start_Park_Position := FALSE;
       "gtyp_MPO".x_Park_Position_Reached := FALSE;
   END_IF;
END_FUNCTION_BLOCK

FUNCTION_BLOCK "PRG_Acknowledge"   // FB18, SCL
TITLE = Program Acknowledge
{ S7_Optimized_Access := 'TRUE' }
AUTHOR : A.Schaefer
VERSION : 0.0
   VAR
      lx_Init : Bool;
      li_StepCase : Int;
      lldt_Ack_old : LDT;
      lfb_TON_Wait : TON_TIME;
      lx_Start_TON_Wait : Bool;
   END_VAR
BEGIN
   IF #lx_Init THEN
       #lfb_TON_Wait(IN := #lx_Start_TON_Wait,
                     PT := T#20s);

       CASE #li_StepCase OF

           0:  // Init
               #lx_Start_TON_Wait := FALSE;

               // check whether acknowledgment has been pressed (time stamp changes)
               IF ("gtyp_Interface_Dashboard".Publish.ldt_AcknowledgeButton > #lldt_Ack_old)
                   OR "gtyp_Setup".x_AcknowledgeButton THEN
                   #lldt_Ack_old := "gtyp_Interface_Dashboard".Publish.ldt_AcknowledgeButton;
                   #li_StepCase := 10;
               END_IF;

           10: // acknowledge Errors
               "gtyp_HBW".x_Error := FALSE;
               "gtyp_MPO".x_Error := FALSE;
               "gtyp_SLD".x_Error := FALSE;
               #li_StepCase := 20;

           20: // Reset acknowledge button
               "gtyp_Setup".x_AcknowledgeButton := FALSE;
               #li_StepCase := 0;
               // Statement section ELSE
           ELSE
               ;
       END_CASE;

   ELSE
       #lx_Init := TRUE;
   END_IF;
END_FUNCTION_BLOCK

FUNCTION_BLOCK "PRG_SLD_Ablauf"   // FB19, SCL
TITLE = Program Ablauf SLD
{ S7_Optimized_Access := 'TRUE' }
AUTHOR : A.Schaefer
VERSION : 0.0
   VAR
      lx_Init : Bool;
      lx_Start_TON_Wait : Bool;
      lx_Time_Error : Bool;
      lt_TON_Wait : Time;
      lx_Start_TON_State : Bool;
      ldt_MQTT : Date_And_Time;
      li_Return_LDT : Int;
      li_Lights : Int;
      li_Lights_old : Int;
      lw_ColorValueMin : Word;
      li_CounterActual : Int;
      lx_White : Bool;
      lx_Blue : Bool;
      lx_Red : Bool;
      li_StepCase : Int;
      ls_Color : String;
      lfb_TOF_ConveyerBelt_Out : TOF_TIME;
      lfb_TON_Wait : TON_TIME;
      lfb_TON_Error : TON_TIME;
      lfb_TON_State : TON_TIME;
      lfb_F_Trig_Counter : F_TRIG;
      lfb_R_Trig_Counter : R_TRIG;
   END_VAR
BEGIN
   IF #lx_Init THEN

       // Restart after set Positioning
       IF "gtyp_Setup".x_Color_Sensor_Calibration THEN
           #li_StepCase := 0;
       END_IF;

       // wait time state
       #lfb_TON_State(IN := NOT #lx_Start_TON_State,
                      PT := T#2s);

       // state of the SLD cyclically transmitted to the cloud
       IF (#lfb_TON_State.Q OR (#li_Lights <> #li_Lights_old)) AND NOT #lx_Start_TON_State THEN
           #li_Lights_old := #li_Lights;
           #lx_Start_TON_State := TRUE;
           #li_Return_LDT := RD_SYS_T(#ldt_MQTT);
           "gtyp_Interface_Dashboard".Subscribe.State_SLD.ldt_ts := DT_TO_LDT(#ldt_MQTT);
           "gtyp_Interface_Dashboard".Subscribe.State_SLD.i_code := #li_Lights;
           "gtyp_Interface_Dashboard".Subscribe.State_SLD.s_description := '';
           "gtyp_Interface_Dashboard".Subscribe.State_SLD.s_station := 'sld';
           "gtyp_Interface_Dashboard".Subscribe.State_SLD.s_target := '';
       END_IF;

       // restart wait time state
       IF NOT #lfb_TON_State.Q AND #lx_Start_TON_State THEN
           #lx_Start_TON_State := FALSE;
       END_IF;

       // FB TON Wait
       #lfb_TON_Wait(IN := #lx_Start_TON_Wait,
                     PT := #lt_TON_Wait);

       // runtime monitoring error
       #lfb_TON_Error(IN := #lx_Time_Error,
                      PT := T#30s);

       // rising edge pulse counter
       #lfb_R_Trig_Counter(CLK := "IX_SLD_PulseCounter_I1");

       // falling edge pulse counter
       #lfb_F_Trig_Counter(CLK := "IX_SLD_PulseCounter_I1");

       // step chain SLD
       CASE #li_StepCase OF

           0:  // Init
               #lx_Start_TON_Wait := FALSE;
               #lx_Time_Error := FALSE;
               #li_Lights := 1;

               IF NOT "gtyp_SLD".x_Error AND NOT "gtyp_Setup".x_Color_Sensor_Calibration THEN
                   #li_StepCase := 10;
               END_IF;

           10: // turn-on Compressor and wait sequence 
               #li_Lights := 2;
               "QX_SLD_Compressor_Q2" := TRUE;

               #lx_Start_TON_Wait := TRUE;
               #lt_TON_Wait := T#1000ms;

               IF #lfb_TON_Wait.Q THEN
                   #lx_Start_TON_Wait := FALSE;
                   #li_StepCase := 20;
               END_IF;

           20:  // reset Ejectors
               "QX_SLD_ValveFirstEjectorWhite_Q3" := FALSE;
               "QX_SLD_ValveSecondEjectorRed_Q4" := FALSE;
               "QX_SLD_ValveThirdEjectorBlue_Q5" := FALSE;
               "QX_SLD_M1_ConveyorBelt_Q1" := FALSE;

               #lx_Start_TON_Wait := TRUE;
               #lt_TON_Wait := T#2000ms;

               IF #lfb_TON_Wait.Q THEN
                   #lx_Start_TON_Wait := FALSE;
                   #li_StepCase := 30;
               END_IF;

           30: // turn-off Compressor 

               "QX_SLD_Compressor_Q2" := FALSE;

               #li_StepCase := 40;

           40: // start belt if Light barrier I2 active

               #li_Lights := 1;
               IF NOT "IX_SLD_LightBarrierInlet_I2" THEN
                   "gtyp_Interface_Dashboard".Subscribe.State_SLD.x_active := TRUE;
                   #li_Lights := 2;
                   "QX_SLD_Compressor_Q2" := TRUE;
                   "QX_SLD_M1_ConveyorBelt_Q1" := TRUE;
                   #lw_ColorValueMin := 40000;
                   #li_CounterActual := 0;
                   #lx_Blue := FALSE;
                   #lx_Red := FALSE;
                   #lx_White := FALSE;
                   #li_StepCase := 50;
               END_IF;

           50: // take the min Value of the Color sensor
               IF #lw_ColorValueMin > "IW_SLD_ColorSensor_A4" THEN
                   #lw_ColorValueMin := "IW_SLD_ColorSensor_A4";
               END_IF;

               #lx_Time_Error := TRUE;

               // Stop when light barrier I3 on 
               IF NOT "IX_SLD_LightBarrierBehindColorSensor_I3" THEN
                   #lx_Time_Error := FALSE;
                   #li_StepCase := 60;
               END_IF;

               // runtime error
               IF #lfb_TON_Error.Q THEN
                   #li_Lights := 4;
                   #lx_Time_Error := FALSE;
                   "QX_SLD_Compressor_Q2" := FALSE;
                   "QX_SLD_M1_ConveyorBelt_Q1" := FALSE;
                   "gtyp_Interface_Dashboard".Subscribe.State_SLD.x_active := FALSE;
                   "gtyp_SLD".x_Error := TRUE;
                   #li_StepCase := 0;
               END_IF;

           60: // analyze color

               IF #lw_ColorValueMin >= "gtyp_SLD".w_Threshold_Red_Blue THEN
                   #lx_Blue := TRUE;
               ELSIF #lw_ColorValueMin <= "gtyp_SLD".w_Threshold_White_Red THEN
                   #lx_White := TRUE;
               ELSIF #lw_ColorValueMin > "gtyp_SLD".w_Threshold_White_Red AND #lw_ColorValueMin < "gtyp_SLD".w_Threshold_Red_Blue THEN
                   #lx_Red := TRUE;
               END_IF;

               // actual counter
               IF #lfb_R_Trig_Counter.Q OR #lfb_F_Trig_Counter.Q THEN
                   #li_CounterActual := #li_CounterActual + 1;
               END_IF;

               // Reached counter value and color set Ejector
               IF (#li_CounterActual = "gtyp_SLD".i_CounterValue_Blue) AND #lx_Blue THEN
                   "QX_SLD_ValveThirdEjectorBlue_Q5" := TRUE;
                   #li_Return_LDT := RD_SYS_T(#ldt_MQTT);
                   "gtyp_SLD".Workpiece.s_state := 'PROCESSED';
                   "gtyp_SLD".History[7].i_code := 700;
                   "gtyp_SLD".History[7].ldt_ts := DT_TO_LDT(#ldt_MQTT);
                   #li_StepCase := 70;
               ELSIF (#li_CounterActual = "gtyp_SLD".i_CounterValue_White) AND #lx_White THEN
                   "QX_SLD_ValveFirstEjectorWhite_Q3" := TRUE;
                   #li_Return_LDT := RD_SYS_T(#ldt_MQTT);
                   "gtyp_SLD".Workpiece.s_state := 'PROCESSED';
                   "gtyp_SLD".History[7].i_code := 700;
                   "gtyp_SLD".History[7].ldt_ts := DT_TO_LDT(#ldt_MQTT);
                   #li_StepCase := 70;
               ELSIF (#li_CounterActual = "gtyp_SLD".i_CounterValue_Red) AND #lx_Red THEN
                   "QX_SLD_ValveSecondEjectorRed_Q4" := TRUE;
                   #li_Return_LDT := RD_SYS_T(#ldt_MQTT);
                   "gtyp_SLD".Workpiece.s_state := 'PROCESSED';
                   "gtyp_SLD".History[7].i_code := 700;
                   "gtyp_SLD".History[7].ldt_ts := DT_TO_LDT(#ldt_MQTT);
                   #li_StepCase := 70;
               ELSIF (#li_CounterActual = 80) THEN
                   #li_Lights := 4;
                   "gtyp_SLD".x_Error := TRUE;
                   #li_StepCase := 70;
               END_IF;

           70: // wait sequence
               #lx_Start_TON_Wait := TRUE;
               #lt_TON_Wait := T#500ms;

               IF #lfb_TON_Wait.Q THEN
                   "QX_SLD_ValveThirdEjectorBlue_Q5" := FALSE;
                   "QX_SLD_ValveFirstEjectorWhite_Q3" := FALSE;
                   "QX_SLD_ValveSecondEjectorRed_Q4" := FALSE;
                   #lx_Start_TON_Wait := FALSE;
                   #li_StepCase := 80;
               END_IF;

           80: // wait sequence

               #lx_Start_TON_Wait := TRUE;
               #lt_TON_Wait := T#2000ms;

               IF #lfb_TON_Wait.Q THEN
                   "QX_SLD_Compressor_Q2" := FALSE;
                   #lx_Start_TON_Wait := FALSE;
                   #li_StepCase := 90;
               END_IF;

           90: // Stop belt
               "QX_SLD_M1_ConveyorBelt_Q1" := FALSE;
               #li_StepCase := 40;
               // Statement section ELSE
           ELSE
               ;
       END_CASE;

   ELSE
       "gtyp_SLD".x_Error := FALSE;
       #li_Lights := 1;
       #lx_Init := TRUE;
   END_IF;
END_FUNCTION_BLOCK

FUNCTION_BLOCK "PRG_Order"   // FB20, SCL
TITLE = Program Order
{ S7_Optimized_Access := 'TRUE' }
AUTHOR : A.Schaefer
VERSION : 0.0
   VAR
      lx_Init : Bool;
      li_StepCase : Int;
      lldt_ts_old : LDT;
      ldt_MQTT : Date_And_Time;
      li_Return_LDT : Int;
      lfb_TON_Wait : TON_TIME;
      lx_Start_TON_Wait : Bool;
   END_VAR
BEGIN
   IF #lx_Init THEN
       #lfb_TON_Wait(IN := #lx_Start_TON_Wait,
                     PT := T#20s);

       // step chain order
       CASE #li_StepCase OF

           0:  // init
               #lx_Start_TON_Wait := FALSE;
               #li_StepCase := 10;

           10: // check whether order button has been pressed (time stamp changes)
               IF ("gtyp_Interface_Dashboard".Publish.OrderWorkpieceButton.ldt_ts > #lldt_ts_old) THEN
                   #li_Return_LDT := RD_SYS_T(#ldt_MQTT);
                   "gtyp_Interface_Dashboard".Subscribe.State_Order.ldt_ts := DT_TO_LDT(#ldt_MQTT);
                   "gtyp_Interface_Dashboard".Subscribe.State_Order.s_state := 'ORDERED';
                   "gtyp_VGR".s_HBW_Outsource_Typ := "gtyp_Interface_Dashboard".Publish.OrderWorkpieceButton.s_type;
                   "gtyp_Interface_Dashboard".Subscribe.State_Order.s_type := "gtyp_VGR".s_HBW_Outsource_Typ;
                   IF "gtyp_VGR".x_Ready_For_Outsource THEN
                       #lldt_ts_old := "gtyp_Interface_Dashboard".Publish.OrderWorkpieceButton.ldt_ts;
                       "gtyp_VGR".x_HBW_Outsource := TRUE;
                       #li_StepCase := 20;
                   END_IF;
               END_IF;

           20: // delete
               IF "gtyp_VGR".x_HBW_PickedUp OR NOT "gtyp_VGR".x_HBW_Outsource THEN
                   "gtyp_VGR".x_HBW_Outsource := FALSE;
                   "gtyp_VGR".s_HBW_Outsource_Typ := '';
                   #li_StepCase := 0;
               END_IF;

               // Statement section ELSE
           ELSE
               ;
       END_CASE;

   ELSE
       #lx_Init := TRUE;
       #lldt_ts_old := LDT#1970-01-01-00:00:00;
   END_IF;
END_FUNCTION_BLOCK

FUNCTION_BLOCK "PRG_SSC_Light"   // FB21, SCL
TITLE = Program Lights
{ S7_Optimized_Access := 'TRUE' }
AUTHOR : A.Schaefer
VERSION : 0.0
   VAR
      lx_Init : Bool;
      lx_Start : Bool;
      li_StepCase : Int;
      ldt_MQTT : Date_And_Time;
      lldt_ts_old : LDT;
      li_Return_LDT : Int;
      lfb_TOF_Camera : TOF_TIME;
      lfb_TON_Schritt : TON_TIME;
      lfb_blinker_cam : "FB_Blinker";
      lfb_blinker_config : "FB_Blinker";
      lx_StartTimer : Bool;
   END_VAR
BEGIN
   IF #lx_Init THEN

       // if camera sen picture - Red light flash
       IF "gtyp_Interface_Dashboard".Subscribe.CameraPicture.ldt_ts > #lldt_ts_old THEN
           #lldt_ts_old := "gtyp_Interface_Dashboard".Subscribe.CameraPicture.ldt_ts;
           #lfb_blinker_cam(int_periodendauer := T#50ms);
       END_IF;

       // reload flash
       "QX_SSC_LED_Red_Online_Q8" := #lfb_blinker_cam.outx_blinker;

       // FB flash config
       #lfb_blinker_config(int_periodendauer := T#500ms);

       //  Deciding which state
       //  Setup - Calibration State
       IF "gtyp_Setup".x_Set_Pos_Activ OR "gtyp_Setup".x_Color_Sensor_Calibration
           OR "gtyp_Setup".x_Counter_Value_Calibration
           OR "gtyp_Setup".x_Clean_Rack_HBW THEN
           "QX_SSC_LED_Green_Q5" := #lfb_blinker_config.outx_blinker;
           "QX_SSC_LED_Yellow_Q6" := #lfb_blinker_config.outx_blinker;
           "QX_SSC_LED_Red_Q7" := #lfb_blinker_config.outx_blinker;
           //  Error State
       ELSIF ("gtyp_Interface_Dashboard".Subscribe.State_HBW.i_code = 4)
           OR ("gtyp_Interface_Dashboard".Subscribe.State_MPO.i_code = 4)
           OR ("gtyp_Interface_Dashboard".Subscribe.State_SLD.i_code = 4)
           OR ("gtyp_Interface_Dashboard".Subscribe.State_VGR.i_code = 4) THEN
           "QX_SSC_LED_Green_Q5" := FALSE;
           "QX_SSC_LED_Yellow_Q6" := FALSE;
           "QX_SSC_LED_Red_Q7" := TRUE;
           //  Proccessing State
       ELSIF ("gtyp_Interface_Dashboard".Subscribe.State_HBW.i_code = 2)
           OR ("gtyp_Interface_Dashboard".Subscribe.State_MPO.i_code = 2)
           OR ("gtyp_Interface_Dashboard".Subscribe.State_SLD.i_code = 2)
           OR ("gtyp_Interface_Dashboard".Subscribe.State_VGR.i_code = 2) THEN
           "QX_SSC_LED_Green_Q5" := FALSE;
           "QX_SSC_LED_Yellow_Q6" := TRUE;
           "QX_SSC_LED_Red_Q7" := FALSE;
           //  Idle State
       ELSIF ("gtyp_Interface_Dashboard".Subscribe.State_HBW.i_code = 1)
           AND ("gtyp_Interface_Dashboard".Subscribe.State_MPO.i_code = 1)
           AND ("gtyp_Interface_Dashboard".Subscribe.State_SLD.i_code = 1)
           AND ("gtyp_Interface_Dashboard".Subscribe.State_VGR.i_code = 1) THEN
           "QX_SSC_LED_Green_Q5" := TRUE;
           "QX_SSC_LED_Yellow_Q6" := FALSE;
           "QX_SSC_LED_Red_Q7" := FALSE;
           //  nothing State
       ELSE
           "QX_SSC_LED_Green_Q5" := FALSE;
           "QX_SSC_LED_Yellow_Q6" := FALSE;
           "QX_SSC_LED_Red_Q7" := FALSE;
       END_IF;


   ELSE
       #lx_Init := TRUE;
   END_IF;
END_FUNCTION_BLOCK

FUNCTION_BLOCK "FB_Axis"   // FB22, SCL
TITLE = Functionblock Axis
{ S7_Optimized_Access := 'TRUE' }
AUTHOR : A.Schaefer
VERSION : 0.0
   VAR_INPUT
      ini_Axis : Int;
      indi_Increment : DInt;
      inx_Ref_Switch : Bool;
      inx_Start_Positioning : Bool;
      inx_Referencing : Bool;
      ini_PWM : Int;
      indi_Target_Position : DInt;
   END_VAR
   VAR_OUTPUT
      outx_Referenced : Bool;
      outx_Position_Reached : Bool;
      outx_Motor_Pos : Bool;
      outx_Motor_Neg : Bool;
      outi_Motor_PWM : Int;
      outdi_Actual_Position : DInt;
   END_VAR
   VAR_IN_OUT
      inouttyp_Config : "typ_Axis_Data";
      inouttyp_Setup : "typ_SetupAxis";
   END_VAR
   VAR
      li_StepCaseSetup : Int;
      li_StepCase : Int;
      lx_Init : Bool;
      lx_Motor_Neg : Bool;
      lx_Motor_Pos : Bool;
      lx_Start_TON_Wait : Bool;
      li_PWM : Int;
      ldi_ValueStep : DInt;
      ldi_Actual_Position : DInt;
      ldi_Actual_Position_Old : DInt;
      lfb_R_Trig_Setup : R_TRIG;
      lfb_R_Trig_Referencing : R_TRIG;
      lfb_TON_Wait : TON_TIME;
   END_VAR
BEGIN
   IF #lx_Init THEN

       // rising edge set up axis
       #lfb_R_Trig_Setup(CLK := #inouttyp_Setup.x_Setup_Activ);

       //Reload when switching to set up
       IF #lfb_R_Trig_Setup.Q THEN
           #inouttyp_Setup.di_LoopValue := #inouttyp_Config.di_Loop_Value;
           #inouttyp_Setup.di_Ref_Pos :=
           #inouttyp_Setup.di_Actual_Ref_Pos := #inouttyp_Config.di_Ref_Pos;
           #inouttyp_Setup.di_Soft_End_Pos_Neg :=
           #inouttyp_Setup.di_Actual_Soft_End_Pos_Neg := #inouttyp_Config.di_Neg_Soft_Switch;
           #inouttyp_Setup.di_Soft_End_Pos_Pos :=
           #inouttyp_Setup.di_Actual_Soft_End_Pos_Pos := #inouttyp_Config.di_Pos_Soft_Switch;
           #inouttyp_Setup.i_PWM := #ini_PWM;
           #inouttyp_Setup.x_Approach_Ref_Pos := FALSE;
           #inouttyp_Setup.x_Approach_Target_Pos := FALSE;
           #inouttyp_Setup.x_Axis_Neg := FALSE;
           #inouttyp_Setup.x_Axis_Pos := FALSE;
           #inouttyp_Setup.x_Set_Ref_Pos := FALSE;
           #inouttyp_Setup.x_Set_Soft_End_Pos := FALSE;
       END_IF;

       #ldi_Actual_Position := #indi_Increment;

       //rising edge referencing
       #lfb_R_Trig_Referencing(CLK := #inx_Referencing);

       //waiting period
       #lfb_TON_Wait(IN := #lx_Start_TON_Wait,
                     PT := T#200ms);

       (**********************************)
       (******   set up step chain   *****)
       (**********************************)
       IF #inouttyp_Setup.i_AxisSelection = #ini_Axis AND #inouttyp_Setup.x_Setup_Activ THEN
           IF #inouttyp_Setup.x_Approach_Ref_Pos THEN
               #inouttyp_Setup.i_Function := 10;
           END_IF;

           CASE #inouttyp_Setup.i_Function OF

               0:  // automatic
                   #ldi_Actual_Position_Old := 0;
                   #inouttyp_Setup.x_Approach_Ref_Pos := FALSE;
                   #lx_Start_TON_Wait := FALSE;

               10: // homing
                   IF #inouttyp_Setup.x_Approach_Ref_Pos THEN
                       IF NOT #inx_Ref_Switch THEN
                           #lx_Motor_Neg := TRUE;
                           #lx_Motor_Pos := FALSE;
                           #outx_Referenced := FALSE;
                       END_IF;

                       IF #inx_Ref_Switch THEN
                           #lx_Motor_Neg := TRUE;
                           #lx_Motor_Pos := TRUE;

                           IF #ldi_Actual_Position = #inouttyp_Config.di_Ref_Pos THEN
                               #inouttyp_Setup.x_Approach_Ref_Pos := FALSE;
                               #lx_Motor_Neg := FALSE;
                               #lx_Motor_Pos := FALSE;
                               #outx_Referenced := TRUE;
                           END_IF;
                       END_IF;
                   END_IF;

               20:  // tap
                   #lx_Motor_Neg := #inouttyp_Setup.x_Axis_Neg AND NOT #inx_Ref_Switch AND NOT (#ldi_Actual_Position <= #inouttyp_Setup.di_Soft_End_Pos_Neg);
                   #lx_Motor_Pos := #inouttyp_Setup.x_Axis_Pos AND NOT #lx_Motor_Neg AND NOT (#ldi_Actual_Position >= #inouttyp_Setup.di_Soft_End_Pos_Pos);

               30:  // tap with increment
                   #ldi_Actual_Position_Old := #ldi_Actual_Position;

                   // positiv
                   IF #inouttyp_Setup.x_Axis_Pos AND NOT ((#ldi_Actual_Position + #inouttyp_Setup.w_Increment + #inouttyp_Setup.di_LoopValue) >= #inouttyp_Setup.di_Soft_End_Pos_Pos) THEN
                       #lx_Motor_Neg := FALSE;
                       #lx_Motor_Pos := TRUE;
                       #ldi_ValueStep := #ldi_Actual_Position_Old + #inouttyp_Setup.w_Increment;

                       // without loop
                       IF (#inouttyp_Setup.di_LoopValue = 0) THEN
                           #inouttyp_Setup.i_Function := 36;
                       ELSE
                           #inouttyp_Setup.i_Function := 31;
                       END_IF;
                       // negativ
                   ELSIF #inouttyp_Setup.x_Axis_Neg AND NOT ((#ldi_Actual_Position - #inouttyp_Setup.w_Increment) <= #inouttyp_Config.di_Neg_Soft_Switch) THEN
                       #lx_Motor_Neg := TRUE;
                       #lx_Motor_Pos := FALSE;
                       #ldi_ValueStep := #ldi_Actual_Position_Old - #inouttyp_Setup.w_Increment;
                       #inouttyp_Setup.i_Function := 34;
                   END_IF;

               31: // with loop
                   IF ((#ldi_Actual_Position >= (#ldi_ValueStep + #inouttyp_Setup.di_LoopValue - #inouttyp_Config.di_Pos_Window)) = 0) THEN
                       #lx_Motor_Neg := TRUE;
                       #lx_Motor_Pos := TRUE;
                       #inouttyp_Setup.i_Function := 32;
                   END_IF;

               32: // wait sequence
                   #lx_Start_TON_Wait := TRUE;

                   IF #lfb_TON_Wait.Q THEN
                       #lx_Motor_Neg := FALSE;
                       #lx_Motor_Pos := FALSE;
                       #lx_Start_TON_Wait := FALSE;
                       #inouttyp_Setup.i_Function := 33;
                   END_IF;

               33: // change direction
                   #lx_Motor_Neg := TRUE;
                   #lx_Motor_Pos := FALSE;
                   #inouttyp_Setup.i_Function := 34;

               34: // position reached negativ
                   IF (#ldi_Actual_Position <= (#ldi_ValueStep + #inouttyp_Config.di_Pos_Window))
                       AND (#ldi_Actual_Position >= (#ldi_ValueStep - #inouttyp_Config.di_Pos_Window)) THEN
                       #lx_Motor_Neg := TRUE;
                       #lx_Motor_Pos := TRUE;
                       #inouttyp_Setup.i_Function := 35;
                   END_IF;

               35: // wait sequence
                   #lx_Start_TON_Wait := TRUE;

                   IF #lfb_TON_Wait.Q THEN
                       #lx_Motor_Neg := FALSE;
                       #lx_Motor_Pos := FALSE;
                       #lx_Start_TON_Wait := FALSE;
                       #inouttyp_Setup.x_Axis_Neg := FALSE;
                       #inouttyp_Setup.x_Axis_Pos := FALSE;
                       #inouttyp_Setup.i_Function := 30;
                   END_IF;


               36: // position reached positiv
                   IF (#ldi_Actual_Position <= (#ldi_ValueStep + #inouttyp_Config.di_Pos_Window))
                       AND (#ldi_Actual_Position >= (#ldi_ValueStep - #inouttyp_Config.di_Pos_Window)) THEN
                       #lx_Motor_Neg := TRUE;
                       #lx_Motor_Pos := TRUE;
                       #inouttyp_Setup.i_Function := 37;
                   END_IF;

               37: // wait sequence
                   #lx_Start_TON_Wait := TRUE;

                   IF #lfb_TON_Wait.Q THEN
                       #lx_Motor_Neg := FALSE;
                       #lx_Motor_Pos := FALSE;
                       #lx_Start_TON_Wait := FALSE;
                       #inouttyp_Setup.x_Axis_Neg := FALSE;
                       #inouttyp_Setup.x_Axis_Pos := FALSE;
                       #inouttyp_Setup.i_Function := 30;
                   END_IF;

               40: // approach position
                   IF #inouttyp_Setup.x_Approach_Target_Pos THEN
                       // positiv
                       IF (#inouttyp_Setup.di_Target_Position > #ldi_Actual_Position) AND NOT ((#inouttyp_Setup.di_Target_Position + #inouttyp_Setup.di_LoopValue) >= #inouttyp_Setup.di_Soft_End_Pos_Pos) THEN
                           #lx_Motor_Neg := FALSE;
                           #lx_Motor_Pos := TRUE;
                           // without loop
                           IF (#inouttyp_Setup.di_LoopValue = 0) THEN
                               #inouttyp_Setup.i_Function := 46;
                           ELSE
                               #inouttyp_Setup.i_Function := 41;
                           END_IF;
                           // negativ
                       ELSIF ((#inouttyp_Setup.di_Target_Position < #ldi_Actual_Position) AND NOT (#inouttyp_Setup.di_Target_Position <= #inouttyp_Config.di_Neg_Soft_Switch)) THEN
                           #lx_Motor_Neg := TRUE;
                           #lx_Motor_Pos := FALSE;
                           #inouttyp_Setup.i_Function := 44;
                       ELSIF (#inouttyp_Setup.di_Target_Position = #ldi_Actual_Position) THEN
                           #inouttyp_Setup.i_Function := 46;
                       END_IF;

                   END_IF;

               41: // with loop
                   IF (#ldi_Actual_Position >= (#inouttyp_Setup.di_Target_Position + #inouttyp_Setup.di_LoopValue - #inouttyp_Config.di_Pos_Window)) THEN
                       #lx_Motor_Neg := TRUE;
                       #lx_Motor_Pos := TRUE;
                       #inouttyp_Setup.i_Function := 42;
                   END_IF;

               42: // wait sequence
                   #lx_Start_TON_Wait := TRUE;

                   IF #lfb_TON_Wait.Q THEN
                       #lx_Motor_Neg := FALSE;
                       #lx_Motor_Pos := FALSE;
                       #lx_Start_TON_Wait := FALSE;
                       #inouttyp_Setup.i_Function := 43;
                   END_IF;

               43: // change direction
                   #lx_Motor_Neg := TRUE;
                   #lx_Motor_Pos := FALSE;
                   #inouttyp_Setup.i_Function := 44;

               44: // position reached negativ
                   IF (#ldi_Actual_Position <= (#inouttyp_Setup.di_Target_Position + #inouttyp_Config.di_Pos_Window))
                       AND (#ldi_Actual_Position >= (#inouttyp_Setup.di_Target_Position - #inouttyp_Config.di_Pos_Window)) THEN
                       #lx_Motor_Neg := TRUE;
                       #lx_Motor_Pos := TRUE;
                       #inouttyp_Setup.i_Function := 45;
                   END_IF;

               45: // wait sequence
                   #lx_Start_TON_Wait := TRUE;

                   IF #lfb_TON_Wait.Q THEN
                       #lx_Motor_Neg := FALSE;
                       #lx_Motor_Pos := FALSE;
                       #lx_Start_TON_Wait := FALSE;
                       #inouttyp_Setup.x_Axis_Neg := FALSE;
                       #inouttyp_Setup.x_Axis_Pos := FALSE;
                       #inouttyp_Setup.i_Function := 40;
                   END_IF;

               46: //  position reached positiv
                   IF (#ldi_Actual_Position <= (#inouttyp_Setup.di_Target_Position + #inouttyp_Config.di_Pos_Window))
                       AND (#ldi_Actual_Position >= (#inouttyp_Setup.di_Target_Position - #inouttyp_Config.di_Pos_Window)) THEN
                       #lx_Motor_Neg := TRUE;
                       #lx_Motor_Pos := TRUE;
                       #inouttyp_Setup.i_Function := 47;
                   END_IF;

               47:  // wait sequence
                   #lx_Start_TON_Wait := TRUE;

                   IF #lfb_TON_Wait.Q THEN
                       #lx_Motor_Neg := FALSE;
                       #lx_Motor_Pos := FALSE;
                       #lx_Start_TON_Wait := FALSE;
                       #inouttyp_Setup.x_Approach_Target_Pos := FALSE;
                       #inouttyp_Setup.i_Function := 40;
                   END_IF;
               ELSE  // Statement section ELSE
                   ;
           END_CASE;

           // set reference point
           IF #inouttyp_Setup.x_Set_Ref_Pos THEN
               #inouttyp_Setup.di_Actual_Ref_Pos :=
               #inouttyp_Config.di_Ref_Pos := #inouttyp_Setup.di_Ref_Pos;
               #inouttyp_Setup.x_Set_Ref_Pos := FALSE;
           END_IF;

           // set software end position
           IF #inouttyp_Setup.x_Set_Soft_End_Pos THEN
               #inouttyp_Setup.di_Actual_Soft_End_Pos_Neg :=
               #inouttyp_Config.di_Neg_Soft_Switch := #inouttyp_Setup.di_Soft_End_Pos_Neg;
               #inouttyp_Setup.di_Actual_Soft_End_Pos_Pos :=
               #inouttyp_Config.di_Pos_Soft_Switch := #inouttyp_Setup.di_Soft_End_Pos_Pos;
               #inouttyp_Setup.x_Set_Soft_End_Pos := FALSE;
           END_IF;

           // reload PWM
           #li_PWM := #inouttyp_Setup.i_PWM;

           // reload actual position
           #inouttyp_Setup.di_ActualPosition := #ldi_Actual_Position;

           (************************************)
           (******   position step chain   *****)
           (************************************)
       ELSIF NOT #inouttyp_Setup.x_Setup_Activ THEN

           // rising edge set up axis
           IF #lfb_R_Trig_Referencing.Q THEN
               #li_StepCase := 0;
           END_IF;

           CASE #li_StepCase OF

               0:  // init
                   #lx_Start_TON_Wait := FALSE;

                   IF #inx_Referencing THEN
                       #li_StepCase := 10;
                       #outx_Position_Reached := FALSE;
                       #outx_Referenced := FALSE;
                   ELSIF #inx_Start_Positioning THEN
                       #li_StepCase := 20;
                       #outx_Position_Reached := FALSE;
                   END_IF;

               10: // homing
                   IF NOT #inx_Ref_Switch THEN
                       #lx_Motor_Neg := TRUE;
                       #lx_Motor_Pos := FALSE;
                   END_IF;

                   IF #inx_Ref_Switch THEN
                       #lx_Motor_Neg := TRUE;
                       #lx_Motor_Pos := TRUE;

                       IF #inx_Ref_Switch THEN
                           IF #ldi_Actual_Position = #inouttyp_Config.di_Ref_Pos THEN
                               #lx_Motor_Neg := FALSE;
                               #lx_Motor_Pos := FALSE;
                               #outx_Referenced := TRUE;
                               #li_StepCase := 11;
                           END_IF;
                       END_IF;
                   END_IF;

               11: // wait not referencing
                   IF NOT #inx_Referencing THEN
                       #li_StepCase := 0;
                   END_IF;

               20: // approach position
                   // positiv
                   IF (#indi_Target_Position > #ldi_Actual_Position) AND NOT ((#indi_Target_Position + #inouttyp_Config.di_Loop_Value) >= #inouttyp_Config.di_Pos_Soft_Switch) THEN
                       #lx_Motor_Neg := FALSE;
                       #lx_Motor_Pos := TRUE;
                       //without loop
                       IF (#inouttyp_Config.di_Loop_Value = 0) THEN
                           #li_StepCase := 26;
                       ELSE
                           #li_StepCase := 21;
                       END_IF;
                       // negativ
                   ELSIF ((#indi_Target_Position < #ldi_Actual_Position) AND NOT (#indi_Target_Position <= #inouttyp_Config.di_Neg_Soft_Switch)) THEN
                       #lx_Motor_Neg := TRUE;
                       #lx_Motor_Pos := FALSE;
                       #li_StepCase := 24;
                   ELSIF (#indi_Target_Position = #ldi_Actual_Position) THEN
                       #li_StepCase := 26;
                   END_IF;

               21: // with loop
                   IF (#ldi_Actual_Position >= (#indi_Target_Position + #inouttyp_Config.di_Loop_Value - #inouttyp_Config.di_Pos_Window)) THEN
                       #lx_Motor_Neg := TRUE;
                       #lx_Motor_Pos := TRUE;
                       #li_StepCase := 22;
                   END_IF;

               22: // wait sequence
                   #lx_Start_TON_Wait := TRUE;

                   IF #lfb_TON_Wait.Q THEN
                       #lx_Motor_Neg := FALSE;
                       #lx_Motor_Pos := FALSE;
                       #lx_Start_TON_Wait := FALSE;
                       #inouttyp_Setup.i_Function := 23;
                   END_IF;

               23: // change direction
                   #lx_Motor_Neg := TRUE;
                   #lx_Motor_Pos := FALSE;
                   #li_StepCase := 24;

               24: // position reached negativ
                   IF (#ldi_Actual_Position <= (#indi_Target_Position + #inouttyp_Config.di_Pos_Window))
                       AND (#ldi_Actual_Position >= (#indi_Target_Position - #inouttyp_Config.di_Pos_Window)) THEN
                       #lx_Motor_Neg := TRUE;
                       #lx_Motor_Pos := TRUE;
                       #li_StepCase := 25;
                   END_IF;

               25: // wait sequence
                   #lx_Start_TON_Wait := TRUE;

                   IF #lfb_TON_Wait.Q THEN
                       #lx_Motor_Neg := FALSE;
                       #lx_Motor_Pos := FALSE;
                       #lx_Start_TON_Wait := FALSE;
                       #outx_Position_Reached := TRUE;
                       #li_StepCase := 28;
                   END_IF;

               26: // position reached positiv
                   IF (#ldi_Actual_Position <= (#indi_Target_Position + #inouttyp_Config.di_Pos_Window))
                       AND (#ldi_Actual_Position >= (#indi_Target_Position - #inouttyp_Config.di_Pos_Window)) THEN
                       #lx_Motor_Neg := TRUE;
                       #lx_Motor_Pos := TRUE;
                       #li_StepCase := 27;
                   END_IF;

               27: // wait sequence
                   #lx_Start_TON_Wait := TRUE;

                   IF #lfb_TON_Wait.Q THEN
                       #lx_Motor_Neg := FALSE;
                       #lx_Motor_Pos := FALSE;
                       #lx_Start_TON_Wait := FALSE;
                       #outx_Position_Reached := TRUE;
                       #li_StepCase := 28;
                   END_IF;

               28: // wait not start positioning
                   IF NOT #inx_Start_Positioning THEN
                       #li_StepCase := 0;
                   END_IF;
                   // statement section ELSE    
               ELSE
                   ;
           END_CASE;

           // reload PWM
           #li_PWM := #ini_PWM;
       END_IF;

       // reload outputs
       #outx_Motor_Neg := #lx_Motor_Neg;
       #outx_Motor_Pos := #lx_Motor_Pos;
       #outi_Motor_PWM := #li_PWM;
       #outdi_Actual_Position := #ldi_Actual_Position;

   ELSE
       #lx_Init := TRUE;
   END_IF;
END_FUNCTION_BLOCK

FUNCTION_BLOCK "PRG_SSC_Axis_Horizontal"   // FB23, SCL
TITLE = Program Axis horizontal SSC
{ S7_Optimized_Access := 'TRUE' }
AUTHOR : A.Schaefer
VERSION : 0.0
   VAR
      lx_Init : Bool;
      lfb_Horizontal_Axis : "FB_Axis";
   END_VAR
BEGIN
   IF #lx_Init THEN

       // FB Axis horizontal
       #lfb_Horizontal_Axis(ini_Axis := 4,
                            indi_Increment := "gtyp_SSC".Horizontal_Axis.di_Increment,
                            inx_Ref_Switch := "IX_SSC_RefSwitchHorizontalAxis_I2",
                            inx_Referencing := "gtyp_SSC".Horizontal_Axis.x_Reference,
                            inx_Start_Positioning := "gtyp_SSC".Horizontal_Axis.x_Start_Positioning,
                            indi_Target_Position := "gtyp_SSC".Horizontal_Axis.di_Target_Position,
                            ini_PWM := "gtyp_SSC".Horizontal_Axis.i_PWM,
                            inouttyp_Config := "gtyp_SSC".Horizontal_Axis.Config,
                            inouttyp_Setup := "gtyp_SetupAxis");

       "QX_SSC_M2_HorizontalAxisCounterclockwise_Q4" := #lfb_Horizontal_Axis.outx_Motor_Neg;
       "QX_SSC_M2_HorizontalAxisClockwise_Q3" := #lfb_Horizontal_Axis.outx_Motor_Pos;
       "QW_SSC_PWM_Horizontal_M2" := #lfb_Horizontal_Axis.outi_Motor_PWM;
       "gtyp_SSC".Horizontal_Axis.di_Actual_Position := #lfb_Horizontal_Axis.outdi_Actual_Position;
       "gtyp_SSC".Horizontal_Axis.x_Referenced := #lfb_Horizontal_Axis.outx_Referenced;
       "gtyp_SSC".Horizontal_Axis.x_Position_Reached := #lfb_Horizontal_Axis.outx_Position_Reached;
   ELSE
       #lx_Init := TRUE;
   END_IF;
END_FUNCTION_BLOCK

FUNCTION_BLOCK "PRG_SSC_Axis_Horizontal_Act_Pos"   // FB24, SCL
TITLE = Program Axis horizontal Actual Position SSC
{ S7_Optimized_Access := 'TRUE' }
AUTHOR : A.Schaefer
VERSION : 0.0
   VAR
      lfb_IN_DEC : "FB_INC_DEC";
   END_VAR
BEGIN
   // FB increment axis
   #lfb_IN_DEC(inx_CHa := "IX_SSC_EncoderHorizontalAxisImp1_B3",
               inx_CHb := "IX_SSC_EncoderHorizontalAxisImp2_B4",
               ini_Ref_Wert := DINT_TO_INT("gtyp_SSC".Horizontal_Axis.Config.di_Ref_Pos),
               inx_RST := "IX_SSC_RefSwitchHorizontalAxis_I2");

   "gtyp_SSC".Horizontal_Axis.di_Increment := #lfb_IN_DEC.outi_cnt;
END_FUNCTION_BLOCK

FUNCTION_BLOCK "PRG_SSC_Axis_Vertical_Act_Pos"   // FB25, SCL
TITLE = Program Axis vertical Actual Position SSC
{ S7_Optimized_Access := 'TRUE' }
AUTHOR : A.Schaefer
VERSION : 0.0
   VAR
      lfb_IN_DEC : "FB_INC_DEC";
   END_VAR
BEGIN
   // FB increment axis
   #lfb_IN_DEC(inx_CHa := "IX_SSC_EncoderVerticalAxisImp2_B2",
               inx_CHb := "IX_SSC_EncoderVerticalAxisImp1_B1",
               ini_Ref_Wert := DINT_TO_INT("gtyp_SSC".Vertical_Axis.Config.di_Ref_Pos),
               inx_RST := "IX_SSC_RefSwitchVerticalAxis_I1");

   "gtyp_SSC".Vertical_Axis.di_Increment := #lfb_IN_DEC.outi_cnt;
END_FUNCTION_BLOCK

FUNCTION_BLOCK "PRG_HBW_Axis_Horizontal_Act_Pos"   // FB26, SCL
TITLE = Program Axis horizontal Actual Position
{ S7_Optimized_Access := 'TRUE' }
AUTHOR : A.Schaefer
VERSION : 0.0
   VAR
      lfb_IN_DEC : "FB_INC_DEC";
   END_VAR
BEGIN
   // FB increment axis
   #lfb_IN_DEC(inx_CHa := "IX_HBW_EncoderHorizontalAxisImp2_B2",
               inx_CHb := "IX_HBW_EncoderHorizontalAxisImp1_B1",
               ini_Ref_Wert := DINT_TO_INT("gtyp_HBW".Horizontal_Axis.Config.di_Ref_Pos),
               inx_RST := "IX_HBW_RefSwitchHorizontalAxis_I1");

   "gtyp_HBW".Horizontal_Axis.di_Increment := #lfb_IN_DEC.outi_cnt;
END_FUNCTION_BLOCK

FUNCTION_BLOCK "PRG_HBW_Axis_Vertical_Act_Pos"   // FB27, SCL
TITLE = Program Axis vertical Actual Position
{ S7_Optimized_Access := 'TRUE' }
AUTHOR : A.Schaefer
VERSION : 0.0
   VAR
      lfb_IN_DEC : "FB_INC_DEC";
   END_VAR
BEGIN
   // FB increment axis
   #lfb_IN_DEC(inx_CHa := "IX_HBW_EncoderVerticalAxisImp1_B3",
               inx_CHb := "IX_HBW_EncoderVerticalAxisImp2_B4",
               ini_Ref_Wert := DINT_TO_INT("gtyp_HBW".Vertical_Axis.Config.di_Ref_Pos),
               inx_RST := "IX_HBW_RefSwitchVerticalAxis_I4");

   "gtyp_HBW".Vertical_Axis.di_Increment := #lfb_IN_DEC.outi_cnt;
END_FUNCTION_BLOCK

FUNCTION_BLOCK "PRG_VGR_Axis_vertical_Act_Pos"   // FB28, SCL
TITLE = Program Axis vertical Actual Position VGR
{ S7_Optimized_Access := 'TRUE' }
AUTHOR : A.Schaefer
VERSION : 0.0
   VAR
      lfb_IN_DEC : "FB_INC_DEC";
   END_VAR
BEGIN
   // FB increment axis
   #lfb_IN_DEC(inx_CHa := "IX_VGR_EncoderVerticalAxisImp1_B1",
               inx_CHb := "IX_VGR_EncoderVerticalAxisImp2_B2",
               ini_Ref_Wert := DINT_TO_INT("gtyp_VGR".vertical_Axis.Config.di_Ref_Pos),
               inx_RST := "IX_VGR_RefSwitchVerticalAxis_I1");

   "gtyp_VGR".vertical_Axis.di_Increment := #lfb_IN_DEC.outi_cnt;
END_FUNCTION_BLOCK

FUNCTION_BLOCK "PRG_VGR_Axis_horizontal_Act_Pos"   // FB29, SCL
TITLE = Program Axis horizontal Actual Position VGR
{ S7_Optimized_Access := 'TRUE' }
AUTHOR : A.Schaefer
VERSION : 0.0
   VAR
      lfb_IN_DEC : "FB_INC_DEC";
   END_VAR
BEGIN
   // FB increment axis
   #lfb_IN_DEC(inx_CHa := "IX_VGR_EncoderHorizontalAxisImp1_B3",
               inx_CHb := "IX_VGR_EncoderHorizontalAxisImp2_B4",
               ini_Ref_Wert := DINT_TO_INT("gtyp_VGR".horizontal_Axis.Config.di_Ref_Pos),
               inx_RST := "IX_VGR_RefSwitchHorizontalAxis_I2");

   "gtyp_VGR".horizontal_Axis.di_Increment := #lfb_IN_DEC.outi_cnt;
END_FUNCTION_BLOCK

FUNCTION_BLOCK "PRG_VGR_Axis_rotate_Act_Pos"   // FB30, SCL
TITLE = Program Axis rotate Actual Position VGR
{ S7_Optimized_Access := 'TRUE' }
AUTHOR : A.Schaefer
VERSION : 0.0
   VAR
      lfb_IN_DEC : "FB_INC_DEC";
   END_VAR
BEGIN
   // FB increment axis
   #lfb_IN_DEC(inx_CHa := "IX_VGR_EncoderRotateImp2_B6",
               inx_CHb := "IX_VGR_EncoderRotateImp1_B5",
               ini_Ref_Wert := DINT_TO_INT("gtyp_VGR".rotate_Axis.Config.di_Ref_Pos),
               inx_RST := "IX_VGR_RefSwitchRotate_I3");

   "gtyp_VGR".rotate_Axis.di_Increment := #lfb_IN_DEC.outi_cnt;
END_FUNCTION_BLOCK

FUNCTION_BLOCK "PRG_HBW_Set_Positioning"   // FB31, SCL
TITLE = Program Set Positioning HBW
{ S7_Optimized_Access := 'TRUE' }
AUTHOR : A.Schaefer
VERSION : 0.0
   VAR
      lx_Init : Bool;
      lx_Start_TON_Wait : Bool;
      lx_Start_Positioning_m : Bool;
      lx_Start_FinalPositioning_m : Bool;
      lx_Start_Offset_m : Bool;
      lt_TON_Wait : Time;
      li_Counter_Hor : Int;
      li_Counter_Ver : Int;
      li_Counter_Act_Hor : Int;
      li_Counter_Act_Ver : Int;
      li_Counter : Int;
      li_StepCase : Int;
      ldi_Pos_Horizontal : DInt;
      ldi_Pos_Vertical : DInt;
      ldi_Offset_Vertical : DInt;
      lfb_R_Trig_Deaktivate : R_TRIG;
      lfb_TON_Wait : TON_TIME;
   END_VAR
BEGIN
   IF #lx_Init THEN

       // FB TON Wait
       #lfb_TON_Wait(IN := #lx_Start_TON_Wait,
                     PT := #lt_TON_Wait);

       #lfb_R_Trig_Deaktivate(CLK := NOT "gtyp_Setup".x_Set_Pos_Activ
                              OR NOT (("gtyp_Setup".i_Pos_Selection > 20)
                              AND ("gtyp_Setup".i_Pos_Selection < 41)));
       // Deaktivate step 110   
       IF #lfb_R_Trig_Deaktivate.Q THEN
           "gtyp_HBW".Horizontal_Axis.x_Start_Positioning := FALSE;
           "gtyp_HBW".Vertical_Axis.x_Start_Positioning := FALSE;
           "gtyp_HBW".Horizontal_Axis.x_Reference := FALSE;
           "gtyp_HBW".Vertical_Axis.x_Reference := FALSE;
           "gtyp_Setup".x_Start_Positioning := FALSE;
           "gtyp_Setup".x_Final_Positioning := FALSE;
           "gtyp_Setup".x_Home_Positioning := FALSE;
           "gtyp_Setup".x_Start_Offset := FALSE;
           "QX_HBW_M4_CantileverBackward_Q8" := FALSE;
           "QX_HBW_M4_CantileverForward_Q7" := FALSE;
           IF (#li_StepCase > 10) THEN
               #li_StepCase := 110;
           END_IF;
       END_IF;

       // Set Positioning activ?
       IF "gtyp_Setup".x_Set_Pos_Activ
           AND (("gtyp_Setup".i_Pos_Selection > 20)
           AND ("gtyp_Setup".i_Pos_Selection < 41))
           AND ((#li_StepCase = 40)
           OR (#li_StepCase = 60)
           OR (#li_StepCase = 80)
           OR (#li_StepCase = 100)) THEN

           // Deciding which Position
           // Position - Belt
           IF "gtyp_Setup".i_Pos_Selection = 21 THEN
               #ldi_Pos_Horizontal := "gtyp_HBW".di_PosBelt_Horizontal;
               #ldi_Pos_Vertical := "gtyp_HBW".di_PosBelt_Vertical;
               #ldi_Offset_Vertical := "gtyp_HBW".di_Offset_Pos_Belt_Vertical;
               // Position - A1 
           ELSIF "gtyp_Setup".i_Pos_Selection = 22 THEN
               #ldi_Pos_Horizontal := "gtyp_HBW".di_PosRack_A1_Horizontal;
               #ldi_Pos_Vertical := "gtyp_HBW".di_PosRack_A1_Vertical;
               #ldi_Offset_Vertical := "gtyp_HBW".di_Offset_Pos_Rack_Vertical;
               // Position - B2 
           ELSIF "gtyp_Setup".i_Pos_Selection = 23 THEN
               #ldi_Pos_Horizontal := "gtyp_HBW".di_PosRack_B2_Horizontal;
               #ldi_Pos_Vertical := "gtyp_HBW".di_PosRack_B2_Vertical;
               #ldi_Offset_Vertical := "gtyp_HBW".di_Offset_Pos_Rack_Vertical;
               // Position - C3 
           ELSIF "gtyp_Setup".i_Pos_Selection = 24 THEN
               #ldi_Pos_Horizontal := "gtyp_HBW".di_PosRack_C3_Horizontal;
               #ldi_Pos_Vertical := "gtyp_HBW".di_PosRack_C3_Vertical;
               #ldi_Offset_Vertical := "gtyp_HBW".di_Offset_Pos_Rack_Vertical;
           END_IF;
       END_IF;

       // Set Positioning activ?
       IF NOT "gtyp_Setup".x_Set_Pos_Activ THEN
           "gtyp_Setup".i_Pos_Selection := 0;
       END_IF;

       // step chain HBW
       CASE #li_StepCase OF

           0:  // init
               #lx_Start_TON_Wait := FALSE;
               #li_StepCase := 10;

           10:  // Set Positioning activ?
               IF "gtyp_Setup".x_Set_Pos_Activ
                   AND (("gtyp_Setup".i_Pos_Selection > 20)
                   AND ("gtyp_Setup".i_Pos_Selection < 41)) THEN

                   "gtyp_HBW".Horizontal_Axis.x_Start_Positioning := FALSE;
                   "gtyp_HBW".Vertical_Axis.x_Start_Positioning := FALSE;
                   "gtyp_HBW".Horizontal_Axis.x_Reference := FALSE;
                   "gtyp_HBW".Vertical_Axis.x_Reference := FALSE;
                   "gtyp_Setup".x_Start_Positioning := FALSE;
                   "gtyp_Setup".x_Final_Positioning := FALSE;
                   "gtyp_Setup".x_Home_Positioning := FALSE;
                   "gtyp_Setup".x_Start_Offset := FALSE;
                   "QX_HBW_M4_CantileverBackward_Q8" := FALSE;
                   "QX_HBW_M4_CantileverForward_Q7" := FALSE;
                   #li_StepCase := 20;
               END_IF;

           20: //homing vertical/horizontal axis

               "gtyp_HBW".Horizontal_Axis.x_Reference := TRUE;
               "gtyp_HBW".Vertical_Axis.x_Reference := TRUE;

               IF NOT "gtyp_HBW".Horizontal_Axis.x_Referenced AND NOT "gtyp_HBW".Vertical_Axis.x_Referenced THEN
                   #li_StepCase := 30;
               END_IF;

           30: // homed vertical/horizontal axis
               IF "gtyp_HBW".Horizontal_Axis.x_Referenced THEN
                   "gtyp_HBW".Horizontal_Axis.x_Reference := FALSE;
               END_IF;
               IF "gtyp_HBW".Vertical_Axis.x_Referenced THEN
                   "gtyp_HBW".Vertical_Axis.x_Reference := FALSE;
               END_IF;

               IF "gtyp_HBW".Horizontal_Axis.x_Referenced AND "gtyp_HBW".Vertical_Axis.x_Referenced THEN
                   "gtyp_HBW".Horizontal_Axis.x_Reference := FALSE;
                   "gtyp_HBW".Vertical_Axis.x_Reference := FALSE;
                   #li_StepCase := 40;
               END_IF;

           40: // Start Positioning Step next
               IF "gtyp_Setup".x_Start_Positioning OR #lx_Start_Positioning_m OR #lx_Start_FinalPositioning_m OR #lx_Start_Offset_m THEN
                   #lx_Start_Positioning_m := FALSE;
                   #li_StepCase := 50;
               END_IF;

           50: // Position vertical/horizontal HBW
               "gtyp_HBW".Horizontal_Axis.di_Target_Position := #ldi_Pos_Horizontal;
               "gtyp_HBW".Horizontal_Axis.x_Start_Positioning := TRUE;
               "gtyp_HBW".Vertical_Axis.di_Target_Position := #ldi_Pos_Vertical;
               "gtyp_HBW".Vertical_Axis.x_Start_Positioning := TRUE;

               IF ("gtyp_HBW".Horizontal_Axis.di_Actual_Position <= (#ldi_Pos_Horizontal + "gtyp_HBW".Horizontal_Axis.Config.di_Pos_Window))
                   AND ("gtyp_HBW".Horizontal_Axis.di_Actual_Position >= (#ldi_Pos_Horizontal - "gtyp_HBW".Horizontal_Axis.Config.di_Pos_Window))
                   AND "gtyp_HBW".Horizontal_Axis.x_Position_Reached THEN
                   "gtyp_HBW".Horizontal_Axis.x_Start_Positioning := FALSE;
               END_IF;

               IF ("gtyp_HBW".Vertical_Axis.di_Actual_Position <= (#ldi_Pos_Vertical + "gtyp_HBW".Vertical_Axis.Config.di_Pos_Window))
                   AND ("gtyp_HBW".Vertical_Axis.di_Actual_Position >= (#ldi_Pos_Vertical - "gtyp_HBW".Vertical_Axis.Config.di_Pos_Window))
                   AND "gtyp_HBW".Vertical_Axis.x_Position_Reached THEN
                   "gtyp_HBW".Vertical_Axis.x_Start_Positioning := FALSE;
               END_IF;

               IF ("gtyp_HBW".Horizontal_Axis.di_Actual_Position <= (#ldi_Pos_Horizontal + "gtyp_HBW".Horizontal_Axis.Config.di_Pos_Window))
                   AND ("gtyp_HBW".Horizontal_Axis.di_Actual_Position >= (#ldi_Pos_Horizontal - "gtyp_HBW".Horizontal_Axis.Config.di_Pos_Window))
                   AND "gtyp_HBW".Horizontal_Axis.x_Position_Reached
                   AND ("gtyp_HBW".Vertical_Axis.di_Actual_Position <= (#ldi_Pos_Vertical + "gtyp_HBW".Vertical_Axis.Config.di_Pos_Window))
                   AND ("gtyp_HBW".Vertical_Axis.di_Actual_Position >= (#ldi_Pos_Vertical - "gtyp_HBW".Vertical_Axis.Config.di_Pos_Window))
                   AND "gtyp_HBW".Vertical_Axis.x_Position_Reached THEN
                   "gtyp_HBW".Horizontal_Axis.x_Start_Positioning := FALSE;
                   "gtyp_HBW".Vertical_Axis.x_Start_Positioning := FALSE;
                   "gtyp_Setup".x_Start_Positioning := FALSE;
                   #li_StepCase := 60;
               END_IF;

           60: // Deciding which doing

               // Start new Positioning
               IF "gtyp_Setup".x_Start_Positioning THEN
                   #lx_Start_Positioning_m := TRUE;
                   #li_StepCase := 10;
                   // Start Final Positioning
               ELSIF "gtyp_Setup".x_Final_Positioning OR #lx_Start_FinalPositioning_m OR #lx_Start_Offset_m THEN
                   #lx_Start_FinalPositioning_m := FALSE;
                   #li_StepCase := 70;
                   // Deaktivate Set Positioning
               ELSIF #lfb_R_Trig_Deaktivate.Q OR "gtyp_Setup".x_Home_Positioning THEN
                   "gtyp_Setup".x_Home_Positioning := FALSE;
                   #li_StepCase := 110;
               END_IF;

           70: // Final Positioning - Cantilever Forward

               "QX_HBW_M4_CantileverBackward_Q8" := FALSE;
               "QX_HBW_M4_CantileverForward_Q7" := TRUE;

               IF "IX_HBW_SwitchCantileverFront_I5" AND NOT "IX_HBW_SwitchCantileverBack_I6" THEN
                   "QX_HBW_M4_CantileverBackward_Q8" := FALSE;
                   "QX_HBW_M4_CantileverForward_Q7" := FALSE;
                   "gtyp_Setup".x_Final_Positioning := FALSE;
                   #li_StepCase := 80;
               END_IF;

           80: // Deciding which doing

               // Start new Positioning
               IF "gtyp_Setup".x_Start_Positioning THEN
                   #lx_Start_Positioning_m := TRUE;
                   #li_StepCase := 110;
                   // Start Final Positioning
               ELSIF "gtyp_Setup".x_Final_Positioning THEN
                   #lx_Start_FinalPositioning_m := TRUE;
                   #li_StepCase := 110;
                   // Start Final Positioning
               ELSIF "gtyp_Setup".x_Start_Offset OR #lx_Start_Offset_m THEN
                   #lx_Start_Offset_m := FALSE;
                   #li_StepCase := 90;
                   // Deaktivate Set Positioning
               ELSIF #lfb_R_Trig_Deaktivate.Q OR "gtyp_Setup".x_Home_Positioning THEN
                   "gtyp_Setup".x_Home_Positioning := FALSE;
                   #li_StepCase := 110;
               END_IF;

           90: // Position vertical+offset HBW
               "gtyp_HBW".Vertical_Axis.di_Target_Position := #ldi_Pos_Vertical - #ldi_Offset_Vertical;
               "gtyp_HBW".Vertical_Axis.x_Start_Positioning := TRUE;

               IF ("gtyp_HBW".Vertical_Axis.di_Actual_Position <= (#ldi_Pos_Vertical - #ldi_Offset_Vertical + "gtyp_HBW".Vertical_Axis.Config.di_Pos_Window))
                   AND ("gtyp_HBW".Vertical_Axis.di_Actual_Position >= (#ldi_Pos_Vertical - #ldi_Offset_Vertical - "gtyp_HBW".Vertical_Axis.Config.di_Pos_Window))
                   AND "gtyp_HBW".Vertical_Axis.x_Position_Reached THEN
                   "gtyp_HBW".Vertical_Axis.x_Start_Positioning := FALSE;
                   "gtyp_Setup".x_Start_Offset := FALSE;
                   #li_StepCase := 100;
               END_IF;

           100: // Deciding which doing

               // Start new Positioning
               IF "gtyp_Setup".x_Start_Positioning THEN
                   #lx_Start_Positioning_m := TRUE;
                   #li_StepCase := 110;
                   // Start Final Positioning
               ELSIF "gtyp_Setup".x_Final_Positioning THEN
                   #lx_Start_FinalPositioning_m := TRUE;
                   #li_StepCase := 110;
                   // Start Final Positioning
               ELSIF "gtyp_Setup".x_Start_Offset THEN
                   #lx_Start_Offset_m := true;
                   #li_StepCase := 110;
                   // Deaktivate Set Positioning
               ELSIF #lfb_R_Trig_Deaktivate.Q OR "gtyp_Setup".x_Home_Positioning THEN
                   "gtyp_Setup".x_Home_Positioning := FALSE;
                   #li_StepCase := 110;
               END_IF;

           110: // Position vertical HBW
               "gtyp_HBW".Vertical_Axis.di_Target_Position := #ldi_Pos_Vertical;
               "gtyp_HBW".Vertical_Axis.x_Start_Positioning := TRUE;

               IF ("gtyp_HBW".Vertical_Axis.di_Actual_Position <= (#ldi_Pos_Vertical + "gtyp_HBW".Vertical_Axis.Config.di_Pos_Window))
                   AND ("gtyp_HBW".Vertical_Axis.di_Actual_Position >= (#ldi_Pos_Vertical - "gtyp_HBW".Vertical_Axis.Config.di_Pos_Window))
                   AND "gtyp_HBW".Vertical_Axis.x_Position_Reached THEN
                   "gtyp_HBW".Vertical_Axis.x_Start_Positioning := FALSE;
                   #li_StepCase := 120;
               END_IF;

           120: // Position vertical Back HBW

               "QX_HBW_M4_CantileverBackward_Q8" := TRUE;
               "QX_HBW_M4_CantileverForward_Q7" := FALSE;

               IF NOT "IX_HBW_SwitchCantileverFront_I5" AND "IX_HBW_SwitchCantileverBack_I6" THEN
                   "QX_HBW_M4_CantileverBackward_Q8" := FALSE;
                   "QX_HBW_M4_CantileverForward_Q7" := FALSE;
                   #li_StepCase := 130;
               END_IF;

           130: // homing vertical/horizontal axis

               "gtyp_HBW".Horizontal_Axis.x_Reference := TRUE;
               "gtyp_HBW".Vertical_Axis.x_Reference := TRUE;

               IF NOT "gtyp_HBW".Horizontal_Axis.x_Referenced AND NOT "gtyp_HBW".Vertical_Axis.x_Referenced THEN
                   #li_StepCase := 140;
               END_IF;

           140: //homed vertical/horizontal axis
               IF "gtyp_HBW".Horizontal_Axis.x_Referenced THEN
                   "gtyp_HBW".Horizontal_Axis.x_Reference := FALSE;
               END_IF;
               IF "gtyp_HBW".Vertical_Axis.x_Referenced THEN
                   "gtyp_HBW".Vertical_Axis.x_Reference := FALSE;
               END_IF;

               IF "gtyp_HBW".Horizontal_Axis.x_Referenced AND "gtyp_HBW".Vertical_Axis.x_Referenced THEN
                   "gtyp_HBW".Horizontal_Axis.x_Reference := FALSE;
                   "gtyp_HBW".Vertical_Axis.x_Reference := FALSE;
                   #li_StepCase := 0;
               END_IF;

               // Statement section ELSE    
           ELSE
               ;
       END_CASE;

       IF (("gtyp_Setup".i_Pos_Selection > 20)
           AND ("gtyp_Setup".i_Pos_Selection < 41)) THEN
           // Reload Pos Value
           "gtyp_Setup".di_Pos_Horizontal := #ldi_Pos_Horizontal;
           "gtyp_Setup".di_Pos_Vertical := #ldi_Pos_Vertical;
           "gtyp_Setup".di_Pos_Rotate := 0;
       END_IF;
   ELSE
       #lx_Init := TRUE;
   END_IF;
END_FUNCTION_BLOCK

FUNCTION_BLOCK "PRG_SSC_Calibration_Color"   // FB32, SCL
TITLE = Program Calibration Color Sensor SSC
{ S7_Optimized_Access := 'TRUE' }
AUTHOR : A.Schaefer
VERSION : 0.0
   VAR
      lx_Init : Bool;
      lx_Start_TON_Wait : Bool;
      lx_Start_Positioning_m : Bool;
      lt_TON_Wait : Time;
      li_StepCase : Int;
      ldi_Pos_Horizontal : DInt;
      ldi_Pos_Vertical : DInt;
      lfb_R_Trig_Deaktivate : R_TRIG;
      lfb_TON_Wait : TON_TIME;
   END_VAR
BEGIN
   IF #lx_Init THEN

       // FB TON Wait
       #lfb_TON_Wait(IN := #lx_Start_TON_Wait,
                     PT := #lt_TON_Wait);

       #lfb_R_Trig_Deaktivate(CLK := NOT "gtyp_Setup".x_Color_Sensor_Calibration
                              OR NOT ("gtyp_Setup".i_Color_Sensor_Selection = 1));
       // Deaktivate step 0   
       IF #lfb_R_Trig_Deaktivate.Q THEN
           "gtyp_Setup".x_Calculate_Value_Color := FALSE;
           "gtyp_Setup".x_Set_Calib_Value_Color_Blue := FALSE;
           "gtyp_Setup".x_Set_Calib_Value_Color_Red := FALSE;
           "gtyp_Setup".x_Set_Calib_Value_Color_White := FALSE;
           "gtyp_Setup".w_Calib_ColorValue_Blue := 0;
           "gtyp_Setup".w_Calib_ColorValue_Red := 0;
           "gtyp_Setup".w_Calib_ColorValue_White := 0;
           "gtyp_Setup".w_Threshold_Red_Blue := 0;
           "gtyp_Setup".w_Threshold_White_Red := 0;
           #li_StepCase := 0;
       END_IF;

       // step chain HBW
       CASE #li_StepCase OF

           0:  // init
               #lx_Start_TON_Wait := FALSE;
               #li_StepCase := 10;

           10:  // Set Calibration activ?
               IF "gtyp_Setup".x_Color_Sensor_Calibration
                   AND ("gtyp_Setup".i_Color_Sensor_Selection = 1) THEN
                   "gtyp_Setup".x_Calculate_Value_Color := FALSE;
                   "gtyp_Setup".x_Set_Calib_Value_Color_Blue := FALSE;
                   "gtyp_Setup".x_Set_Calib_Value_Color_Red := FALSE;
                   "gtyp_Setup".x_Set_Calib_Value_Color_White := FALSE;
                   "gtyp_Setup".w_Calib_ColorValue_Blue := 0;
                   "gtyp_Setup".w_Calib_ColorValue_Red := 0;
                   "gtyp_Setup".w_Calib_ColorValue_White := 0;
                   "gtyp_Setup".w_Threshold_Red_Blue := 0;
                   "gtyp_Setup".w_Threshold_White_Red := 0;
                   #li_StepCase := 20;
               END_IF;

           20: // wait for set Values or Calculate

